LIN {X 0,Y 185.438,Z 182.881,A -85,B 0,C 180,E1 -22182.587,E2 -22182.587} C_VEL
LIN {X 0,Y 186.423,Z 185.682,A -85,B 0,C 180,E1 -22183.112,E2 -22183.112} C_VEL
LIN {X 0,Y 188.894,Z 188.498,A -85,B 0,C 180,E1 -22184.064,E2 -22184.064} C_VEL
LIN {X 0,Y 191.056,Z 191.778,A -85,B 0,C 180,E1 -22184.906,E2 -22184.906} C_VEL
LIN {X 0,Y 192.643,Z 194.162,A -85,B 0,C 180,E1 -22185.503,E2 -22185.503} C_VEL
LIN {X 0,Y 197.521,Z 201.307,A -85,B 0,C 180,E1 -22187.235,E2 -22187.235} C_VEL
LIN {X 0,Y 203.04,Z 210.464,A -85,B 0,C 180,E1 -22189.09,E2 -22189.09} C_VEL
LIN {X 0,Y 209.264,Z 223.651,A -85,B 0,C 180,E1 -22191.133,E2 -22191.133} C_VEL
LIN {X 0,Y 213.51,Z 234.001,A -85,B 0,C 180,E1 -22192.484,E2 -22192.484} C_VEL
LIN {X 0,Y 210.832,Z 286.169,A -85,B 0,C 180,E1 -22194.15,E2 -22194.15} C_VEL
LIN {X 0,Y 209.437,Z 299.447,A -85,B 0,C 180,E1 -22194.897,E2 -22194.897} C_VEL
LIN {X 0,Y 207.404,Z 312.457,A -85,B 0,C 180,E1 -22196.006,E2 -22196.006} C_VEL
LIN {X 0,Y 205.128,Z 323.758,A -85,B 0,C 180,E1 -22197.342,E2 -22197.342} C_VEL
LIN {X 0,Y 202.167,Z 335.393,A -85,B 0,C 180,E1 -22199.152,E2 -22199.152} C_VEL
LIN {X 0,Y 199.074,Z 345.843,A -85,B 0,C 180,E1 -22201.249,E2 -22201.249} C_VEL
LIN {X 0,Y 196.058,Z 355.418,A -85,B 0,C 180,E1 -22203.724,E2 -22203.724} C_VEL
LIN {X 0,Y 193.173,Z 363.626,A -85,B 0,C 180,E1 -22206.409,E2 -22206.409} C_VEL
LIN {X 0,Y 190.261,Z 371.037,A -85,B 0,C 180,E1 -22209.456,E2 -22209.456} C_VEL
LIN {X 0,Y 187.898,Z 376.982,A -85,B 0,C 180,E1 -22212.589,E2 -22212.589} C_VEL
LIN {X 0,Y 186.02,Z 381.679,A -85,B 0,C 180,E1 -22215.784,E2 -22215.784} C_VEL
LIN {X 0,Y 184.706,Z 385.27,A -85,B 0,C 180,E1 -22219.033,E2 -22219.033} C_VEL
LIN {X 0,Y 184.105,Z 387.123,A -85,B 0,C 180,E1 -22221.217,E2 -22221.217} C_VEL
LIN {X 0,Y 183.397,Z 389.328,A -85,B 0,C 180,E1 -22225.109,E2 -22225.109} C_VEL
LIN {X 0,Y 183.186,Z 390.114,A -85,B 0,C 180,E1 -22227.801,E2 -22227.801} C_VEL
LIN {X 0,Y 183.146,Z 390.342,A -85,B 0,C 180,E1 -22230,E2 -22230} C_VEL
LIN {X 0,Y 183.184,Z 390.147,A -85,B 0,C 180,E1 -22232.199,E2 -22232.199} C_VEL
LIN {X 0,Y 183.618,Z 388.592,A -85,B 0,C 180,E1 -22236.593,E2 -22236.593} C_VEL
LIN {X 0,Y 184.036,Z 387.234,A -85,B 0,C 180,E1 -22238.786,E2 -22238.786} C_VEL
LIN {X 0,Y 185.055,Z 384.362,A -85,B 0,C 180,E1 -22242.056,E2 -22242.056} C_VEL
LIN {X 0,Y 186.565,Z 380.465,A -85,B 0,C 180,E1 -22245.289,E2 -22245.289} C_VEL
LIN {X 0,Y 188.562,Z 375.438,A -85,B 0,C 180,E1 -22248.47,E2 -22248.47} C_VEL
LIN {X 0,Y 191.128,Z 369.103,A -85,B 0,C 180,E1 -22251.574,E2 -22251.574} C_VEL
LIN {X 0,Y 194.162,Z 361.178,A -85,B 0,C 180,E1 -22254.599,E2 -22254.599} C_VEL
LIN {X 0,Y 196.883,Z 353.061,A -85,B 0,C 180,E1 -22257.086,E2 -22257.086} C_VEL
LIN {X 0,Y 200.037,Z 343.242,A -85,B 0,C 180,E1 -22259.463,E2 -22259.463} C_VEL
LIN {X 0,Y 202.839,Z 333.532,A -85,B 0,C 180,E1 -22261.313,E2 -22261.313} C_VEL
LIN {X 0,Y 205.421,Z 323.01,A -85,B 0,C 180,E1 -22262.896,E2 -22262.896} C_VEL
LIN {X 0,Y 207.938,Z 310.339,A -85,B 0,C 180,E1 -22264.334,E2 -22264.334} C_VEL
LIN {X 0,Y 209.725,Z 297.869,A -85,B 0,C 180,E1 -22265.364,E2 -22265.364} C_VEL
LIN {X 0,Y 211.06,Z 284.908,A -85,B 0,C 180,E1 -22266.034,E2 -22266.034} C_VEL
LIN {X 0,Y 213.59,Z 233.928,A -85,B 0,C 180,E1 -22267.668,E2 -22267.668} C_VEL
LIN {X 0,Y 207.958,Z 220.601,A -85,B 0,C 180,E1 -22269.464,E2 -22269.464} C_VEL
LIN {X 0,Y 201.794,Z 208.024,A -85,B 0,C 180,E1 -22271.512,E2 -22271.512} C_VEL
LIN {X 0,Y 195.962,Z 198.988,A -85,B 0,C 180,E1 -22273.494,E2 -22273.494} C_VEL
LIN {X 0,Y 193.215,Z 194.973,A -85,B 0,C 180,E1 -22274.48,E2 -22274.48} C_VEL
LIN {X 0,Y 190.972,Z 191.674,A -85,B 0,C 180,E1 -22275.321,E2 -22275.321} C_VEL
LIN {X 0,Y 188.815,Z 188.335,A -85,B 0,C 180,E1 -22276.17,E2 -22276.17} C_VEL
LIN {X 0,Y 186.181,Z 185.235,A -85,B 0,C 180,E1 -22277.198,E2 -22277.198} C_VEL
LIN {X 0,Y 185.45,Z 182.877,A -85,B 0,C 180,E1 -22277.611,E2 -22277.611} C_VEL
LIN {X 0,Y 185.544,Z 182.862,A -85,B 0,C 180,E1 -22282.696,E2 -22282.696} C_VEL
LIN {X 0,Y 185.545,Z 182.864,A -85,B 0,C 180,E1 -22287.975,E2 -22287.975} C_VEL
LIN {X 0,Y 185.582,Z 182.86,A -85,B 0,C 180,E1 -22290.575,E2 -22290.575} C_VEL
LIN {X 0,Y 185.588,Z 182.867,A -85,B 0,C 180,E1 -22295.382,E2 -22295.382} C_VEL
LIN {X 0,Y 185.675,Z 182.858,A -85,B 0,C 180,E1 -22301.133,E2 -22301.133} C_VEL
LIN {X 0,Y 185.765,Z 182.842,A -85,B 0,C 180,E1 -22306.88,E2 -22306.88} C_VEL
LIN {X 0,Y 186.009,Z 182.795,A -85,B 0,C 180,E1 -22311.307,E2 -22311.307} C_VEL
LIN {X 0,Y 186.208,Z 182.773,A -85,B 0,C 180,E1 -22317.837,E2 -22317.837} C_VEL
LIN {X 0,Y 186.405,Z 182.75,A -85,B 0,C 180,E1 -22320,E2 -22320} C_VEL
LIN {X 0,Y 185.924,Z 182.815,A -85,B 0,C 180,E1 -22324.336,E2 -22324.336} C_VEL
LIN {X 0,Y 186.009,Z 182.811,A -85,B 0,C 180,E1 -22328.693,E2 -22328.693} C_VEL
LIN {X 0,Y 185.734,Z 182.829,A -85,B 0,C 180,E1 -22333.122,E2 -22333.122} C_VEL
LIN {X 0,Y 185.689,Z 182.848,A -85,B 0,C 180,E1 -22337.625,E2 -22337.625} C_VEL
LIN {X 0,Y 185.578,Z 182.868,A -85,B 0,C 180,E1 -22342.254,E2 -22342.254} C_VEL
LIN {X 0,Y 185.558,Z 182.869,A -85,B 0,C 180,E1 -22347.033,E2 -22347.033} C_VEL
LIN {X 0,Y 185.577,Z 182.86,A -85,B 0,C 180,E1 -22349.493,E2 -22349.493} C_VEL
LIN {X 0,Y 185.499,Z 182.869,A -85,B 0,C 180,E1 -22354.632,E2 -22354.632} C_VEL
LIN {X 0,Y 185.505,Z 182.874,A -85,B 0,C 180,E1 -22357.313,E2 -22357.313} C_VEL
LIN {X 0,Y 185.495,Z 183.087,A -85,B 0,C 180,E1 -22360.733,E2 -22360.733} C_VEL
LIN {X 0,Y 186.322,Z 185.835,A -85,B 0,C 180,E1 -22362.606,E2 -22362.606} C_VEL
LIN {X 0,Y 189.088,Z 190.333,A -85,B 0,C 180,E1 -22363.748,E2 -22363.748} C_VEL
LIN {X 0,Y 193.463,Z 197.495,A -85,B 0,C 180,E1 -22365.444,E2 -22365.444} C_VEL
LIN {X 0,Y 199.054,Z 207.457,A -85,B 0,C 180,E1 -22367.479,E2 -22367.479} C_VEL
LIN {X 0,Y 205.15,Z 219.677,A -85,B 0,C 180,E1 -22369.566,E2 -22369.566} C_VEL
LIN {X 0,Y 211.223,Z 234.41,A -85,B 0,C 180,E1 -22371.577,E2 -22371.577} C_VEL
LIN {X 0,Y 212.326,Z 238.091,A -85,B 0,C 180,E1 -22371.966,E2 -22371.966} C_VEL
LIN {X 0,Y 213.063,Z 245.558,A -85,B 0,C 180,E1 -22372.431,E2 -22372.431} C_VEL
LIN {X 0,Y 212.354,Z 259.49,A -85,B 0,C 180,E1 -22372.865,E2 -22372.865} C_VEL
LIN {X 0,Y 211.584,Z 265.346,A -85,B 0,C 180,E1 -22372.946,E2 -22372.946} C_VEL
LIN {X 0,Y 205.962,Z 284.372,A -85,B 0,C 180,E1 -22372.571,E2 -22372.571} C_VEL
LIN {X 0,Y 205.095,Z 290.216,A -85,B 0,C 180,E1 -22372.672,E2 -22372.672} C_VEL
LIN {X 0,Y 203.834,Z 303.973,A -85,B 0,C 180,E1 -22373.356,E2 -22373.356} C_VEL
LIN {X 0,Y 201.749,Z 316.536,A -85,B 0,C 180,E1 -22374.304,E2 -22374.304} C_VEL
LIN {X 0,Y 199.213,Z 328.676,A -85,B 0,C 180,E1 -22375.635,E2 -22375.635} C_VEL
LIN {X 0,Y 196.423,Z 339.649,A -85,B 0,C 180,E1 -22377.237,E2 -22377.237} C_VEL
LIN {X 0,Y 192.952,Z 350.849,A -85,B 0,C 180,E1 -22379.341,E2 -22379.341} C_VEL
LIN {X 0,Y 189.536,Z 360.785,A -85,B 0,C 180,E1 -22381.786,E2 -22381.786} C_VEL
LIN {X 0,Y 186.521,Z 368.936,A -85,B 0,C 180,E1 -22384.322,E2 -22384.322} C_VEL
LIN {X 0,Y 183.553,Z 376.941,A -85,B 0,C 180,E1 -22387.488,E2 -22387.488} C_VEL
LIN {X 0,Y 180.921,Z 383.353,A -85,B 0,C 180,E1 -22390.72,E2 -22390.72} C_VEL
LIN {X 0,Y 178.761,Z 388.446,A -85,B 0,C 180,E1 -22394.026,E2 -22394.026} C_VEL
LIN {X 0,Y 177.39,Z 392.408,A -85,B 0,C 180,E1 -22397.414,E2 -22397.414} C_VEL
LIN {X 0,Y 176.468,Z 395.337,A -85,B 0,C 180,E1 -22400.834,E2 -22400.834} C_VEL
LIN {X 0,Y 175.946,Z 397.726,A -85,B 0,C 180,E1 -22405.418,E2 -22405.418} C_VEL
LIN {X 0,Y 175.949,Z 398.335,A -85,B 0,C 180,E1 -22407.711,E2 -22407.711} C_VEL
LIN {X 0,Y 176.022,Z 398.547,A -85,B 0,C 180,E1 -22410,E2 -22410} C_VEL
LIN {X 0,Y 175.947,Z 398.162,A -85,B 0,C 180,E1 -22413.037,E2 -22413.037} C_VEL
LIN {X 0,Y 176.137,Z 396.699,A -85,B 0,C 180,E1 -22416.875,E2 -22416.875} C_VEL
LIN {X 0,Y 176.468,Z 395.291,A -85,B 0,C 180,E1 -22419.167,E2 -22419.167} C_VEL
LIN {X 0,Y 177.39,Z 392.343,A -85,B 0,C 180,E1 -22422.586,E2 -22422.586} C_VEL
LIN {X 0,Y 178.76,Z 388.356,A -85,B 0,C 180,E1 -22425.974,E2 -22425.974} C_VEL
LIN {X 0,Y 181.33,Z 382.235,A -85,B 0,C 180,E1 -22429.824,E2 -22429.824} C_VEL
LIN {X 0,Y 184.328,Z 374.773,A -85,B 0,C 180,E1 -22433.379,E2 -22433.379} C_VEL
LIN {X 0,Y 187.075,Z 367.259,A -85,B 0,C 180,E1 -22436.195,E2 -22436.195} C_VEL
LIN {X 0,Y 190.171,Z 358.756,A -85,B 0,C 180,E1 -22438.713,E2 -22438.713} C_VEL
LIN {X 0,Y 193.689,Z 348.253,A -85,B 0,C 180,E1 -22441.135,E2 -22441.135} C_VEL
LIN {X 0,Y 197.144,Z 336.428,A -85,B 0,C 180,E1 -22443.237,E2 -22443.237} C_VEL
LIN {X 0,Y 200.028,Z 324.506,A -85,B 0,C 180,E1 -22444.816,E2 -22444.816} C_VEL
LIN {X 0,Y 202.45,Z 312.094,A -85,B 0,C 180,E1 -22446.014,E2 -22446.014} C_VEL
LIN {X 0,Y 204.293,Z 299.341,A -85,B 0,C 180,E1 -22446.856,E2 -22446.856} C_VEL
LIN {X 0,Y 205.334,Z 285.462,A -85,B 0,C 180,E1 -22447.419,E2 -22447.419} C_VEL
LIN {X 0,Y 207.266,Z 245.004,A -85,B 0,C 180,E1 -22448.75,E2 -22448.75} C_VEL
LIN {X 0,Y 206.492,Z 239.162,A -85,B 0,C 180,E1 -22449.177,E2 -22449.177} C_VEL
LIN {X 0,Y 201.216,Z 225.726,A -85,B 0,C 180,E1 -22451.022,E2 -22451.022} C_VEL
LIN {X 0,Y 195.205,Z 212.97,A -85,B 0,C 180,E1 -22453.19,E2 -22453.19} C_VEL
LIN {X 0,Y 188.351,Z 200.534,A -85,B 0,C 180,E1 -22455.828,E2 -22455.828} C_VEL
LIN {X 0,Y 183.78,Z 193.268,A -85,B 0,C 180,E1 -22457.716,E2 -22457.716} C_VEL
LIN {X 0,Y 181.859,Z 190.145,A -85,B 0,C 180,E1 -22458.563,E2 -22458.563} C_VEL
LIN {X 0,Y 178.959,Z 185.72,A -85,B 0,C 180,E1 -22459.887,E2 -22459.887} C_VEL
LIN {X 0,Y 178.665,Z 184.95,A -85,B 0,C 180,E1 -22460.267,E2 -22460.267} C_VEL
LIN {X 0,Y 178.412,Z 183.762,A -85,B 0,C 180,E1 -22461.242,E2 -22461.242} C_VEL
LIN {X 0,Y 178.484,Z 183.753,A -85,B 0,C 180,E1 -22466.546,E2 -22466.546} C_VEL
LIN {X 0,Y 178.444,Z 183.752,A -85,B 0,C 180,E1 -22471.796,E2 -22471.796} C_VEL
LIN {X 0,Y 178.516,Z 183.749,A -85,B 0,C 180,E1 -22474.889,E2 -22474.889} C_VEL
LIN {X 0,Y 178.623,Z 183.731,A -85,B 0,C 180,E1 -22480.785,E2 -22480.785} C_VEL
LIN {X 0,Y 178.658,Z 183.724,A -85,B 0,C 180,E1 -22486.348,E2 -22486.348} C_VEL
LIN {X 0,Y 178.912,Z 183.7,A -85,B 0,C 180,E1 -22490.96,E2 -22490.96} C_VEL
LIN {X 0,Y 179.153,Z 183.664,A -85,B 0,C 180,E1 -22497.752,E2 -22497.752} C_VEL
LIN {X 0,Y 179.369,Z 183.629,A -85,B 0,C 180,E1 -22500,E2 -22500} C_VEL
LIN {X 0,Y 178.867,Z 183.694,A -85,B 0,C 180,E1 -22504.507,E2 -22504.507} C_VEL
LIN {X 0,Y 178.912,Z 183.699,A -85,B 0,C 180,E1 -22509.04,E2 -22509.04} C_VEL
LIN {X 0,Y 178.659,Z 183.729,A -85,B 0,C 180,E1 -22513.652,E2 -22513.652} C_VEL
LIN {X 0,Y 178.639,Z 183.731,A -85,B 0,C 180,E1 -22519.23,E2 -22519.23} C_VEL
LIN {X 0,Y 178.535,Z 183.746,A -85,B 0,C 180,E1 -22525.125,E2 -22525.125} C_VEL
LIN {X 0,Y 178.48,Z 183.749,A -85,B 0,C 180,E1 -22530.791,E2 -22530.791} C_VEL
LIN {X 0,Y 178.493,Z 183.752,A -85,B 0,C 180,E1 -22534.223,E2 -22534.223} C_VEL
LIN {X 0,Y 178.43,Z 183.754,A -85,B 0,C 180,E1 -22539.796,E2 -22539.796} C_VEL
LIN {X 0,Y 178.447,Z 183.753,A -85,B 0,C 180,E1 -22540.16,E2 -22540.16} C_VEL
LIN {X 0,Y 179.378,Z 186.499,A -85,B 0,C 180,E1 -22540.684,E2 -22540.684} C_VEL
LIN {X 0,Y 181.415,Z 188.713,A -85,B 0,C 180,E1 -22541.562,E2 -22541.562} C_VEL
LIN {X 0,Y 184.268,Z 192.886,A -85,B 0,C 180,E1 -22542.795,E2 -22542.795} C_VEL
LIN {X 0,Y 185.614,Z 194.718,A -85,B 0,C 180,E1 -22543.346,E2 -22543.346} C_VEL
LIN {X 0,Y 188.82,Z 199.398,A -85,B 0,C 180,E1 -22544.623,E2 -22544.623} C_VEL
LIN {X 0,Y 195.085,Z 208.87,A -85,B 0,C 180,E1 -22546.94,E2 -22546.94} C_VEL
LIN {X 0,Y 199.32,Z 216.409,A -85,B 0,C 180,E1 -22548.433,E2 -22548.433} C_VEL
LIN {X 0,Y 206.254,Z 231.957,A -85,B 0,C 180,E1 -22550.819,E2 -22550.819} C_VEL
LIN {X 0,Y 207.807,Z 235.855,A -85,B 0,C 180,E1 -22551.339,E2 -22551.339} C_VEL
LIN {X 0,Y 205.268,Z 284.588,A -85,B 0,C 180,E1 -22552.926,E2 -22552.926} C_VEL
LIN {X 0,Y 203.962,Z 297.662,A -85,B 0,C 180,E1 -22553.612,E2 -22553.612} C_VEL
LIN {X 0,Y 202.37,Z 308.094,A -85,B 0,C 180,E1 -22554.43,E2 -22554.43} C_VEL
LIN {X 0,Y 199.971,Z 320.431,A -85,B 0,C 180,E1 -22555.784,E2 -22555.784} C_VEL
LIN {X 0,Y 197.266,Z 331.509,A -85,B 0,C 180,E1 -22557.394,E2 -22557.394} C_VEL
LIN {X 0,Y 193.921,Z 342.804,A -85,B 0,C 180,E1 -22559.51,E2 -22559.51} C_VEL
LIN {X 0,Y 190.885,Z 352.098,A -85,B 0,C 180,E1 -22561.777,E2 -22561.777} C_VEL
LIN {X 0,Y 187.801,Z 360.925,A -85,B 0,C 180,E1 -22564.51,E2 -22564.51} C_VEL
LIN {X 0,Y 184.585,Z 368.922,A -85,B 0,C 180,E1 -22567.62,E2 -22567.62} C_VEL
LIN {X 0,Y 181.882,Z 375.338,A -85,B 0,C 180,E1 -22570.826,E2 -22570.826} C_VEL
LIN {X 0,Y 179.745,Z 380.425,A -85,B 0,C 180,E1 -22574.115,E2 -22574.115} C_VEL
LIN {X 0,Y 178.15,Z 384.373,A -85,B 0,C 180,E1 -22577.469,E2 -22577.469} C_VEL
LIN {X 0,Y 177.084,Z 387.286,A -85,B 0,C 180,E1 -22580.866,E2 -22580.866} C_VEL
LIN {X 0,Y 176.568,Z 388.678,A -85,B 0,C 180,E1 -22583.142,E2 -22583.142} C_VEL
LIN {X 0,Y 176.262,Z 389.668,A -85,B 0,C 180,E1 -22585.426,E2 -22585.426} C_VEL
LIN {X 0,Y 176.102,Z 390.276,A -85,B 0,C 180,E1 -22587.713,E2 -22587.713} C_VEL
LIN {X 0,Y 176.058,Z 390.504,A -85,B 0,C 180,E1 -22590,E2 -22590} C_VEL
LIN {X 0,Y 176.1,Z 390.309,A -85,B 0,C 180,E1 -22592.287,E2 -22592.287} C_VEL
LIN {X 0,Y 176.562,Z 388.754,A -85,B 0,C 180,E1 -22596.858,E2 -22596.858} C_VEL
LIN {X 0,Y 177.033,Z 387.395,A -85,B 0,C 180,E1 -22599.137,E2 -22599.137} C_VEL
LIN {X 0,Y 178.12,Z 384.523,A -85,B 0,C 180,E1 -22602.533,E2 -22602.533} C_VEL
LIN {X 0,Y 179.718,Z 380.626,A -85,B 0,C 180,E1 -22605.887,E2 -22605.887} C_VEL
LIN {X 0,Y 181.834,Z 375.599,A -85,B 0,C 180,E1 -22609.179,E2 -22609.179} C_VEL
LIN {X 0,Y 184.544,Z 369.263,A -85,B 0,C 180,E1 -22612.385,E2 -22612.385} C_VEL
LIN {X 0,Y 187.71,Z 361.338,A -85,B 0,C 180,E1 -22615.503,E2 -22615.503} C_VEL
LIN {X 0,Y 190.575,Z 353.263,A -85,B 0,C 180,E1 -22618.046,E2 -22618.046} C_VEL
LIN {X 0,Y 193.884,Z 343.4,A -85,B 0,C 180,E1 -22620.496,E2 -22620.496} C_VEL
LIN {X 0,Y 196.825,Z 333.689,A -85,B 0,C 180,E1 -22622.385,E2 -22622.385} C_VEL
LIN {X 0,Y 199.494,Z 323.167,A -85,B 0,C 180,E1 -22624.004,E2 -22624.004} C_VEL
LIN {X 0,Y 202.127,Z 310.494,A -85,B 0,C 180,E1 -22625.466,E2 -22625.466} C_VEL
LIN {X 0,Y 204.024,Z 297.735,A -85,B 0,C 180,E1 -22626.538,E2 -22626.538} C_VEL
LIN {X 0,Y 205.354,Z 285.32,A -85,B 0,C 180,E1 -22627.187,E2 -22627.187} C_VEL
LIN {X 0,Y 207.85,Z 235.79,A -85,B 0,C 180,E1 -22628.824,E2 -22628.824} C_VEL
LIN {X 0,Y 201.999,Z 221.957,A -85,B 0,C 180,E1 -22630.814,E2 -22630.814} C_VEL
LIN {X 0,Y 196.888,Z 211.745,A -85,B 0,C 180,E1 -22632.613,E2 -22632.613} C_VEL
LIN {X 0,Y 190.234,Z 201.344,A -85,B 0,C 180,E1 -22635.038,E2 -22635.038} C_VEL
LIN {X 0,Y 184.437,Z 193.04,A -85,B 0,C 180,E1 -22637.346,E2 -22637.346} C_VEL
LIN {X 0,Y 182.218,Z 189.939,A -85,B 0,C 180,E1 -22638.293,E2 -22638.293} C_VEL
LIN {X 0,Y 181.458,Z 188.733,A -85,B 0,C 180,E1 -22638.635,E2 -22638.635} C_VEL
LIN {X 0,Y 179.398,Z 186.531,A -85,B 0,C 180,E1 -22639.525,E2 -22639.525} C_VEL
LIN {X 0,Y 178.453,Z 183.756,A -85,B 0,C 180,E1 -22640.118,E2 -22640.118} C_VEL
LIN {X 0,Y 178.496,Z 183.738,A -85,B 0,C 180,E1 -22645.775,E2 -22645.775} C_VEL
LIN {X 0,Y 178.523,Z 183.744,A -85,B 0,C 180,E1 -22650.006,E2 -22650.006} C_VEL
LIN {X 0,Y 178.535,Z 183.746,A -85,B 0,C 180,E1 -22654.875,E2 -22654.875} C_VEL
LIN {X 0,Y 178.624,Z 183.735,A -85,B 0,C 180,E1 -22660.784,E2 -22660.784} C_VEL
LIN {X 0,Y 178.682,Z 183.72,A -85,B 0,C 180,E1 -22666.35,E2 -22666.35} C_VEL
LIN {X 0,Y 178.938,Z 183.675,A -85,B 0,C 180,E1 -22670.961,E2 -22670.961} C_VEL
LIN {X 0,Y 179.154,Z 183.651,A -85,B 0,C 180,E1 -22677.752,E2 -22677.752} C_VEL
LIN {X 0,Y 179.368,Z 183.626,A -85,B 0,C 180,E1 -22680,E2 -22680} C_VEL
LIN {X 0,Y 178.872,Z 183.691,A -85,B 0,C 180,E1 -22684.507,E2 -22684.507} C_VEL
LIN {X 0,Y 178.959,Z 183.692,A -85,B 0,C 180,E1 -22689.038,E2 -22689.038} C_VEL
LIN {X 0,Y 178.666,Z 183.709,A -85,B 0,C 180,E1 -22693.651,E2 -22693.651} C_VEL
LIN {X 0,Y 178.649,Z 183.718,A -85,B 0,C 180,E1 -22698.344,E2 -22698.344} C_VEL
LIN {X 0,Y 178.497,Z 183.749,A -85,B 0,C 180,E1 -22703.187,E2 -22703.187} C_VEL
LIN {X 0,Y 178.485,Z 183.752,A -85,B 0,C 180,E1 -22708.197,E2 -22708.197} C_VEL
LIN {X 0,Y 178.477,Z 183.743,A -85,B 0,C 180,E1 -22710.791,E2 -22710.791} C_VEL
LIN {X 0,Y 178.484,Z 183.743,A -85,B 0,C 180,E1 -22714.219,E2 -22714.219} C_VEL
LIN {X 0,Y 178.417,Z 183.872,A -85,B 0,C 180,E1 -22718.757,E2 -22718.757} C_VEL
LIN {X 0,Y 178.895,Z 185.52,A -85,B 0,C 180,E1 -22719.947,E2 -22719.947} C_VEL
LIN {X 0,Y 181.77,Z 190.049,A -85,B 0,C 180,E1 -22721.278,E2 -22721.278} C_VEL
LIN {X 0,Y 183.051,Z 192.016,A -85,B 0,C 180,E1 -22721.843,E2 -22721.843} C_VEL
LIN {X 0,Y 187.094,Z 198.569,A -85,B 0,C 180,E1 -22723.559,E2 -22723.559} C_VEL
LIN {X 0,Y 191.402,Z 205.843,A -85,B 0,C 180,E1 -22725.269,E2 -22725.269} C_VEL
LIN {X 0,Y 197.565,Z 217.59,A -85,B 0,C 180,E1 -22727.574,E2 -22727.574} C_VEL
LIN {X 0,Y 203.143,Z 230.178,A -85,B 0,C 180,E1 -22729.563,E2 -22729.563} C_VEL
LIN {X 0,Y 206.773,Z 239.68,A -85,B 0,C 180,E1 -22730.828,E2 -22730.828} C_VEL
LIN {X 0,Y 207.444,Z 245.987,A -85,B 0,C 180,E1 -22731.252,E2 -22731.252} C_VEL
LIN {X 0,Y 205.095,Z 290.216,A -85,B 0,C 180,E1 -22732.672,E2 -22732.672} C_VEL
LIN {X 0,Y 204.558,Z 294.107,A -85,B 0,C 180,E1 -22732.764,E2 -22732.764} C_VEL
LIN {X 0,Y 202.211,Z 301.678,A -85,B 0,C 180,E1 -22732.816,E2 -22732.816} C_VEL
LIN {X 0,Y 196.875,Z 314.527,A -85,B 0,C 180,E1 -22733.032,E2 -22733.032} C_VEL
LIN {X 0,Y 195.298,Z 320.024,A -85,B 0,C 180,E1 -22733.452,E2 -22733.452} C_VEL
LIN {X 0,Y 192.536,Z 331.95,A -85,B 0,C 180,E1 -22734.907,E2 -22734.907} C_VEL
LIN {X 0,Y 189.274,Z 343.502,A -85,B 0,C 180,E1 -22736.792,E2 -22736.792} C_VEL
LIN {X 0,Y 185.763,Z 353.904,A -85,B 0,C 180,E1 -22738.971,E2 -22738.971} C_VEL
LIN {X 0,Y 182.615,Z 362.41,A -85,B 0,C 180,E1 -22741.245,E2 -22741.245} C_VEL
LIN {X 0,Y 179.56,Z 370.262,A -85,B 0,C 180,E1 -22743.875,E2 -22743.875} C_VEL
LIN {X 0,Y 176.475,Z 377.933,A -85,B 0,C 180,E1 -22747.152,E2 -22747.152} C_VEL
LIN {X 0,Y 173.385,Z 385.01,A -85,B 0,C 180,E1 -22751.079,E2 -22751.079} C_VEL
LIN {X 0,Y 171.351,Z 389.717,A -85,B 0,C 180,E1 -22754.538,E2 -22754.538} C_VEL
LIN {X 0,Y 170.053,Z 393.318,A -85,B 0,C 180,E1 -22758.075,E2 -22758.075} C_VEL
LIN {X 0,Y 169.427,Z 395.174,A -85,B 0,C 180,E1 -22760.449,E2 -22760.449} C_VEL
LIN {X 0,Y 168.86,Z 397.564,A -85,B 0,C 180,E1 -22765.225,E2 -22765.225} C_VEL
LIN {X 0,Y 168.858,Z 398.173,A -85,B 0,C 180,E1 -22767.615,E2 -22767.615} C_VEL
LIN {X 0,Y 168.934,Z 398.385,A -85,B 0,C 180,E1 -22770,E2 -22770} C_VEL
LIN {X 0,Y 168.85,Z 398.109,A -85,B 0,C 180,E1 -22772.627,E2 -22772.627} C_VEL
LIN {X 0,Y 169.072,Z 396.536,A -85,B 0,C 180,E1 -22777.164,E2 -22777.164} C_VEL
LIN {X 0,Y 169.427,Z 395.128,A -85,B 0,C 180,E1 -22779.551,E2 -22779.551} C_VEL
LIN {X 0,Y 170.436,Z 392.179,A -85,B 0,C 180,E1 -22783.109,E2 -22783.109} C_VEL
LIN {X 0,Y 171.92,Z 388.192,A -85,B 0,C 180,E1 -22786.628,E2 -22786.628} C_VEL
LIN {X 0,Y 174.637,Z 382.071,A -85,B 0,C 180,E1 -22790.618,E2 -22790.618} C_VEL
LIN {X 0,Y 177.485,Z 375.379,A -85,B 0,C 180,E1 -22793.95,E2 -22793.95} C_VEL
LIN {X 0,Y 180.691,Z 367.093,A -85,B 0,C 180,E1 -22797.195,E2 -22797.195} C_VEL
LIN {X 0,Y 183.952,Z 358.59,A -85,B 0,C 180,E1 -22799.78,E2 -22799.78} C_VEL
LIN {X 0,Y 187.638,Z 348.087,A -85,B 0,C 180,E1 -22802.258,E2 -22802.258} C_VEL
LIN {X 0,Y 191.245,Z 336.262,A -85,B 0,C 180,E1 -22804.403,E2 -22804.403} C_VEL
LIN {X 0,Y 194.236,Z 324.338,A -85,B 0,C 180,E1 -22806.013,E2 -22806.013} C_VEL
LIN {X 0,Y 196.743,Z 311.924,A -85,B 0,C 180,E1 -22807.231,E2 -22807.231} C_VEL
LIN {X 0,Y 198.665,Z 299.183,A -85,B 0,C 180,E1 -22808.081,E2 -22808.081} C_VEL
LIN {X 0,Y 199.793,Z 284.339,A -85,B 0,C 180,E1 -22808.687,E2 -22808.687} C_VEL
LIN {X 0,Y 201.734,Z 246.08,A -85,B 0,C 180,E1 -22809.965,E2 -22809.965} C_VEL
LIN {X 0,Y 201.101,Z 241.562,A -85,B 0,C 180,E1 -22810.321,E2 -22810.321} C_VEL
LIN {X 0,Y 195.466,Z 227.242,A -85,B 0,C 180,E1 -22812.421,E2 -22812.421} C_VEL
LIN {X 0,Y 189.097,Z 214.028,A -85,B 0,C 180,E1 -22814.887,E2 -22814.887} C_VEL
LIN {X 0,Y 183.283,Z 203.692,A -85,B 0,C 180,E1 -22817.294,E2 -22817.294} C_VEL
LIN {X 0,Y 178.309,Z 195.507,A -85,B 0,C 180,E1 -22819.537,E2 -22819.537} C_VEL
LIN {X 0,Y 174.548,Z 189.931,A -85,B 0,C 180,E1 -22821.354,E2 -22821.354} C_VEL
LIN {X 0,Y 172.188,Z 187.163,A -85,B 0,C 180,E1 -22822.525,E2 -22822.525} C_VEL
LIN {X 0,Y 171.415,Z 184.96,A -85,B 0,C 180,E1 -22823.065,E2 -22823.065} C_VEL
LIN {X 0,Y 171.381,Z 184.637,A -85,B 0,C 180,E1 -22823.515,E2 -22823.515} C_VEL
LIN {X 0,Y 171.418,Z 184.632,A -85,B 0,C 180,E1 -22829.427,E2 -22829.427} C_VEL
LIN {X 0,Y 171.444,Z 184.628,A -85,B 0,C 180,E1 -22834.402,E2 -22834.402} C_VEL
LIN {X 0,Y 171.579,Z 184.606,A -85,B 0,C 180,E1 -22840.872,E2 -22840.872} C_VEL
LIN {X 0,Y 171.577,Z 184.61,A -85,B 0,C 180,E1 -22845.773,E2 -22845.773} C_VEL
LIN {X 0,Y 171.849,Z 184.579,A -85,B 0,C 180,E1 -22850.585,E2 -22850.585} C_VEL
LIN {X 0,Y 171.817,Z 184.578,A -85,B 0,C 180,E1 -22855.308,E2 -22855.308} C_VEL
LIN {X 0,Y 172.332,Z 184.505,A -85,B 0,C 180,E1 -22860,E2 -22860} C_VEL
LIN {X 0,Y 171.815,Z 184.57,A -85,B 0,C 180,E1 -22864.693,E2 -22864.693} C_VEL
LIN {X 0,Y 171.849,Z 184.577,A -85,B 0,C 180,E1 -22869.415,E2 -22869.415} C_VEL
LIN {X 0,Y 171.58,Z 184.612,A -85,B 0,C 180,E1 -22874.227,E2 -22874.227} C_VEL
LIN {X 0,Y 171.559,Z 184.615,A -85,B 0,C 180,E1 -22879.575,E2 -22879.575} C_VEL
LIN {X 0,Y 171.47,Z 184.626,A -85,B 0,C 180,E1 -22885.617,E2 -22885.617} C_VEL
LIN {X 0,Y 171.443,Z 184.626,A -85,B 0,C 180,E1 -22890.587,E2 -22890.587} C_VEL
LIN {X 0,Y 171.403,Z 184.628,A -85,B 0,C 180,E1 -22896.48,E2 -22896.48} C_VEL
LIN {X 0,Y 171.396,Z 184.634,A -85,B 0,C 180,E1 -22897.308,E2 -22897.308} C_VEL
LIN {X 0,Y 172.287,Z 187.267,A -85,B 0,C 180,E1 -22897.891,E2 -22897.891} C_VEL
LIN {X 0,Y 174.275,Z 189.515,A -85,B 0,C 180,E1 -22898.873,E2 -22898.873} C_VEL
LIN {X 0,Y 175.154,Z 190.413,A -85,B 0,C 180,E1 -22899.288,E2 -22899.288} C_VEL
LIN {X 0,Y 177.244,Z 193.633,A -85,B 0,C 180,E1 -22900.311,E2 -22900.311} C_VEL
LIN {X 0,Y 178.639,Z 195.287,A -85,B 0,C 180,E1 -22900.939,E2 -22900.939} C_VEL
LIN {X 0,Y 181.349,Z 199.009,A -85,B 0,C 180,E1 -22902.139,E2 -22902.139} C_VEL
LIN {X 0,Y 189.231,Z 210.901,A -85,B 0,C 180,E1 -22905.356,E2 -22905.356} C_VEL
LIN {X 0,Y 194.301,Z 219.723,A -85,B 0,C 180,E1 -22907.262,E2 -22907.262} C_VEL
LIN {X 0,Y 200.847,Z 234.43,A -85,B 0,C 180,E1 -22909.656,E2 -22909.656} C_VEL
LIN {X 0,Y 202.22,Z 237.907,A -85,B 0,C 180,E1 -22910.146,E2 -22910.146} C_VEL
LIN {X 0,Y 199.625,Z 285.168,A -85,B 0,C 180,E1 -22911.714,E2 -22911.714} C_VEL
LIN {X 0,Y 198.269,Z 298.107,A -85,B 0,C 180,E1 -22912.419,E2 -22912.419} C_VEL
LIN {X 0,Y 196.643,Z 308.264,A -85,B 0,C 180,E1 -22913.227,E2 -22913.227} C_VEL
LIN {X 0,Y 194.154,Z 320.598,A -85,B 0,C 180,E1 -22914.608,E2 -22914.608} C_VEL
LIN {X 0,Y 191.325,Z 331.675,A -85,B 0,C 180,E1 -22916.249,E2 -22916.249} C_VEL
LIN {X 0,Y 187.833,Z 342.97,A -85,B 0,C 180,E1 -22918.411,E2 -22918.411} C_VEL
LIN {X 0,Y 184.405,Z 352.935,A -85,B 0,C 180,E1 -22920.928,E2 -22920.928} C_VEL
LIN {X 0,Y 180.88,Z 362.568,A -85,B 0,C 180,E1 -22924.08,E2 -22924.08} C_VEL
LIN {X 0,Y 177.552,Z 370.253,A -85,B 0,C 180,E1 -22927.298,E2 -22927.298} C_VEL
LIN {X 0,Y 174.356,Z 377.31,A -85,B 0,C 180,E1 -22931.188,E2 -22931.188} C_VEL
LIN {X 0,Y 172.277,Z 382.006,A -85,B 0,C 180,E1 -22934.623,E2 -22934.623} C_VEL
LIN {X 0,Y 170.764,Z 385.596,A -85,B 0,C 180,E1 -22938.125,E2 -22938.125} C_VEL
LIN {X 0,Y 170.069,Z 387.449,A -85,B 0,C 180,E1 -22940.485,E2 -22940.485} C_VEL
LIN {X 0,Y 169.526,Z 388.841,A -85,B 0,C 180,E1 -22942.856,E2 -22942.856} C_VEL
LIN {X 0,Y 169.007,Z 390.439,A -85,B 0,C 180,E1 -22947.617,E2 -22947.617} C_VEL
LIN {X 0,Y 168.972,Z 390.666,A -85,B 0,C 180,E1 -22950,E2 -22950} C_VEL
LIN {X 0,Y 169.134,Z 390.063,A -85,B 0,C 180,E1 -22954.229,E2 -22954.229} C_VEL
LIN {X 0,Y 169.52,Z 388.915,A -85,B 0,C 180,E1 -22957.145,E2 -22957.145} C_VEL
LIN {X 0,Y 170.01,Z 387.557,A -85,B 0,C 180,E1 -22959.518,E2 -22959.518} C_VEL
LIN {X 0,Y 171.178,Z 384.685,A -85,B 0,C 180,E1 -22963.05,E2 -22963.05} C_VEL
LIN {X 0,Y 172.899,Z 380.787,A -85,B 0,C 180,E1 -22966.531,E2 -22966.531} C_VEL
LIN {X 0,Y 175.141,Z 375.759,A -85,B 0,C 180,E1 -22969.943,E2 -22969.943} C_VEL
LIN {X 0,Y 178.005,Z 369.423,A -85,B 0,C 180,E1 -22973.255,E2 -22973.255} C_VEL
LIN {X 0,Y 181.24,Z 361.694,A -85,B 0,C 180,E1 -22976.401,E2 -22976.401} C_VEL
LIN {X 0,Y 184.334,Z 353.422,A -85,B 0,C 180,E1 -22979.085,E2 -22979.085} C_VEL
LIN {X 0,Y 187.813,Z 343.559,A -85,B 0,C 180,E1 -22981.593,E2 -22981.593} C_VEL
LIN {X 0,Y 190.873,Z 333.847,A -85,B 0,C 180,E1 -22983.525,E2 -22983.525} C_VEL
LIN {X 0,Y 193.655,Z 323.323,A -85,B 0,C 180,E1 -22985.178,E2 -22985.178} C_VEL
LIN {X 0,Y 196.397,Z 310.648,A -85,B 0,C 180,E1 -22986.666,E2 -22986.666} C_VEL
LIN {X 0,Y 198.332,Z 298.219,A -85,B 0,C 180,E1 -22987.731,E2 -22987.731} C_VEL
LIN {X 0,Y 199.731,Z 285.725,A -85,B 0,C 180,E1 -22988.407,E2 -22988.407} C_VEL
LIN {X 0,Y 202.265,Z 237.923,A -85,B 0,C 180,E1 -22990.019,E2 -22990.019} C_VEL
LIN {X 0,Y 197.086,Z 225.556,A -85,B 0,C 180,E1 -22991.893,E2 -22991.893} C_VEL
LIN {X 0,Y 192.557,Z 216.344,A -85,B 0,C 180,E1 -22993.583,E2 -22993.583} C_VEL
LIN {X 0,Y 186.433,Z 206.562,A -85,B 0,C 180,E1 -22995.941,E2 -22995.941} C_VEL
LIN {X 0,Y 180.722,Z 198.314,A -85,B 0,C 180,E1 -22998.337,E2 -22998.337} C_VEL
LIN {X 0,Y 177.858,Z 194.233,A -85,B 0,C 180,E1 -22999.639,E2 -22999.639} C_VEL
LIN {X 0,Y 175.626,Z 191.295,A -85,B 0,C 180,E1 -23000.694,E2 -23000.694} C_VEL
LIN {X 0,Y 174.797,Z 189.854,A -85,B 0,C 180,E1 -23001.121,E2 -23001.121} C_VEL
LIN {X 0,Y 172.586,Z 187.733,A -85,B 0,C 180,E1 -23002.186,E2 -23002.186} C_VEL
LIN {X 0,Y 171.519,Z 185.307,A -85,B 0,C 180,E1 -23002.815,E2 -23002.815} C_VEL
LIN {X 0,Y 171.405,Z 184.623,A -85,B 0,C 180,E1 -23002.971,E2 -23002.971} C_VEL
LIN {X 0,Y 171.428,Z 184.619,A -85,B 0,C 180,E1 -23007.794,E2 -23007.794} C_VEL
LIN {X 0,Y 171.449,Z 184.619,A -85,B 0,C 180,E1 -23010.534,E2 -23010.534} C_VEL
LIN {X 0,Y 171.458,Z 184.624,A -85,B 0,C 180,E1 -23015.801,E2 -23015.801} C_VEL
LIN {X 0,Y 171.58,Z 184.612,A -85,B 0,C 180,E1 -23020.872,E2 -23020.872} C_VEL
LIN {X 0,Y 171.594,Z 184.595,A -85,B 0,C 180,E1 -23025.774,E2 -23025.774} C_VEL
LIN {X 0,Y 171.873,Z 184.556,A -85,B 0,C 180,E1 -23030.586,E2 -23030.586} C_VEL
LIN {X 0,Y 171.823,Z 184.582,A -85,B 0,C 180,E1 -23035.308,E2 -23035.308} C_VEL
LIN {X 0,Y 172.331,Z 184.501,A -85,B 0,C 180,E1 -23040,E2 -23040} C_VEL
LIN {X 0,Y 171.821,Z 184.567,A -85,B 0,C 180,E1 -23044.692,E2 -23044.692} C_VEL
LIN {X 0,Y 171.888,Z 184.573,A -85,B 0,C 180,E1 -23049.413,E2 -23049.413} C_VEL
LIN {X 0,Y 171.593,Z 184.593,A -85,B 0,C 180,E1 -23054.226,E2 -23054.226} C_VEL
LIN {X 0,Y 171.54,Z 184.598,A -85,B 0,C 180,E1 -23059.558,E2 -23059.558} C_VEL
LIN {X 0,Y 171.458,Z 184.613,A -85,B 0,C 180,E1 -23065.609,E2 -23065.609} C_VEL
LIN {X 0,Y 171.44,Z 184.619,A -85,B 0,C 180,E1 -23070.586,E2 -23070.586} C_VEL
LIN {X 0,Y 171.378,Z 184.646,A -85,B 0,C 180,E1 -23076.532,E2 -23076.532} C_VEL
LIN {X 0,Y 171.428,Z 185.016,A -85,B 0,C 180,E1 -23076.84,E2 -23076.84} C_VEL
LIN {X 0,Y 172.371,Z 187.483,A -85,B 0,C 180,E1 -23077.428,E2 -23077.428} C_VEL
LIN {X 0,Y 175.783,Z 191.623,A -85,B 0,C 180,E1 -23079.114,E2 -23079.114} C_VEL
LIN {X 0,Y 179.96,Z 198.211,A -85,B 0,C 180,E1 -23081.106,E2 -23081.106} C_VEL
LIN {X 0,Y 182.934,Z 203.033,A -85,B 0,C 180,E1 -23082.432,E2 -23082.432} C_VEL
LIN {X 0,Y 187.872,Z 211.743,A -85,B 0,C 180,E1 -23084.513,E2 -23084.513} C_VEL
LIN {X 0,Y 193.556,Z 222.981,A -85,B 0,C 180,E1 -23086.754,E2 -23086.754} C_VEL
LIN {X 0,Y 198.813,Z 235.205,A -85,B 0,C 180,E1 -23088.733,E2 -23088.733} C_VEL
LIN {X 0,Y 201.49,Z 242.558,A -85,B 0,C 180,E1 -23089.731,E2 -23089.731} C_VEL
LIN {X 0,Y 201.867,Z 247.666,A -85,B 0,C 180,E1 -23090.053,E2 -23090.053} C_VEL
LIN {X 0,Y 199.159,Z 294.791,A -85,B 0,C 180,E1 -23091.633,E2 -23091.633} C_VEL
LIN {X 0,Y 197.51,Z 308.209,A -85,B 0,C 180,E1 -23092.429,E2 -23092.429} C_VEL
LIN {X 0,Y 195.298,Z 320.024,A -85,B 0,C 180,E1 -23093.452,E2 -23093.452} C_VEL
LIN {X 0,Y 193.625,Z 325.449,A -85,B 0,C 180,E1 -23093.941,E2 -23093.941} C_VEL
LIN {X 0,Y 189.151,Z 334.031,A -85,B 0,C 180,E1 -23094.599,E2 -23094.599} C_VEL
LIN {X 0,Y 184.321,Z 342.221,A -85,B 0,C 180,E1 -23095.472,E2 -23095.472} C_VEL
LIN {X 0,Y 182.121,Z 347.03,A -85,B 0,C 180,E1 -23096.3,E2 -23096.3} C_VEL
LIN {X 0,Y 178.578,Z 356.732,A -85,B 0,C 180,E1 -23098.57,E2 -23098.57} C_VEL
LIN {X 0,Y 175.055,Z 365.549,A -85,B 0,C 180,E1 -23101.199,E2 -23101.199} C_VEL
LIN {X 0,Y 171.941,Z 373.091,A -85,B 0,C 180,E1 -23104.059,E2 -23104.059} C_VEL
LIN {X 0,Y 168.868,Z 380.004,A -85,B 0,C 180,E1 -23107.358,E2 -23107.358} C_VEL
LIN {X 0,Y 166.672,Z 384.849,A -85,B 0,C 180,E1 -23110.286,E2 -23110.286} C_VEL
LIN {X 0,Y 164.484,Z 389.555,A -85,B 0,C 180,E1 -23113.875,E2 -23113.875} C_VEL
LIN {X 0,Y 163.098,Z 393.157,A -85,B 0,C 180,E1 -23117.558,E2 -23117.558} C_VEL
LIN {X 0,Y 162.41,Z 395.012,A -85,B 0,C 180,E1 -23120.032,E2 -23120.032} C_VEL
LIN {X 0,Y 161.763,Z 397.402,A -85,B 0,C 180,E1 -23125.015,E2 -23125.015} C_VEL
LIN {X 0,Y 161.762,Z 398.07,A -85,B 0,C 180,E1 -23127.818,E2 -23127.818} C_VEL
LIN {X 0,Y 161.833,Z 398.223,A -85,B 0,C 180,E1 -23130,E2 -23130} C_VEL
LIN {X 0,Y 161.76,Z 397.996,A -85,B 0,C 180,E1 -23132.49,E2 -23132.49} C_VEL
LIN {X 0,Y 161.999,Z 396.373,A -85,B 0,C 180,E1 -23137.478,E2 -23137.478} C_VEL
LIN {X 0,Y 162.41,Z 394.964,A -85,B 0,C 180,E1 -23139.968,E2 -23139.968} C_VEL
LIN {X 0,Y 163.483,Z 392.015,A -85,B 0,C 180,E1 -23143.677,E2 -23143.677} C_VEL
LIN {X 0,Y 165.111,Z 388.028,A -85,B 0,C 180,E1 -23147.335,E2 -23147.335} C_VEL
LIN {X 0,Y 167.957,Z 381.906,A -85,B 0,C 180,E1 -23151.477,E2 -23151.477} C_VEL
LIN {X 0,Y 171.248,Z 374.532,A -85,B 0,C 180,E1 -23155.238,E2 -23155.238} C_VEL
LIN {X 0,Y 174.383,Z 366.928,A -85,B 0,C 180,E1 -23158.265,E2 -23158.265} C_VEL
LIN {X 0,Y 177.821,Z 358.425,A -85,B 0,C 180,E1 -23160.917,E2 -23160.917} C_VEL
LIN {X 0,Y 181.652,Z 347.921,A -85,B 0,C 180,E1 -23163.458,E2 -23163.458} C_VEL
LIN {X 0,Y 185.421,Z 336.095,A -85,B 0,C 180,E1 -23165.645,E2 -23165.645} C_VEL
LIN {X 0,Y 188.533,Z 324.169,A -85,B 0,C 180,E1 -23167.283,E2 -23167.283} C_VEL
LIN {X 0,Y 191.153,Z 311.754,A -85,B 0,C 180,E1 -23168.516,E2 -23168.516} C_VEL
LIN {X 0,Y 193.193,Z 298.464,A -85,B 0,C 180,E1 -23169.408,E2 -23169.408} C_VEL
LIN {X 0,Y 194.374,Z 282.989,A -85,B 0,C 180,E1 -23170.033,E2 -23170.033} C_VEL
LIN {X 0,Y 196.297,Z 247.155,A -85,B 0,C 180,E1 -23171.248,E2 -23171.248} C_VEL
LIN {X 0,Y 195.732,Z 243.939,A -85,B 0,C 180,E1 -23171.546,E2 -23171.546} C_VEL
LIN {X 0,Y 190.759,Z 231.04,A -85,B 0,C 180,E1 -23173.526,E2 -23173.526} C_VEL
LIN {X 0,Y 184.889,Z 218.615,A -85,B 0,C 180,E1 -23175.941,E2 -23175.941} C_VEL
LIN {X 0,Y 179.468,Z 208.696,A -85,B 0,C 180,E1 -23178.327,E2 -23178.327} C_VEL
LIN {X 0,Y 174.518,Z 200.5,A -85,B 0,C 180,E1 -23180.692,E2 -23180.692} C_VEL
LIN {X 0,Y 171.369,Z 195.583,A -85,B 0,C 180,E1 -23182.315,E2 -23182.315} C_VEL
LIN {X 0,Y 168.882,Z 192.499,A -85,B 0,C 180,E1 -23183.629,E2 -23183.629} C_VEL
LIN {X 0,Y 168.002,Z 190.885,A -85,B 0,C 180,E1 -23184.15,E2 -23184.15} C_VEL
LIN {X 0,Y 165.574,Z 188.727,A -85,B 0,C 180,E1 -23185.483,E2 -23185.483} C_VEL
LIN {X 0,Y 164.446,Z 186.178,A -85,B 0,C 180,E1 -23186.249,E2 -23186.249} C_VEL
LIN {X 0,Y 164.339,Z 185.514,A -85,B 0,C 180,E1 -23186.4,E2 -23186.4} C_VEL
LIN {X 0,Y 164.37,Z 185.51,A -85,B 0,C 180,E1 -23189.13,E2 -23189.13} C_VEL
LIN {X 0,Y 164.395,Z 185.508,A -85,B 0,C 180,E1 -23194.691,E2 -23194.691} C_VEL
LIN {X 0,Y 164.485,Z 185.496,A -85,B 0,C 180,E1 -23200.051,E2 -23200.051} C_VEL
LIN {X 0,Y 164.524,Z 185.492,A -85,B 0,C 180,E1 -23205.149,E2 -23205.149} C_VEL
LIN {X 0,Y 164.769,Z 185.461,A -85,B 0,C 180,E1 -23210.177,E2 -23210.177} C_VEL
LIN {X 0,Y 164.832,Z 185.44,A -85,B 0,C 180,E1 -23212.651,E2 -23212.651} C_VEL
LIN {X 0,Y 165.049,Z 185.422,A -85,B 0,C 180,E1 -23217.56,E2 -23217.56} C_VEL
LIN {X 0,Y 165.294,Z 185.381,A -85,B 0,C 180,E1 -23220,E2 -23220} C_VEL
LIN {X 0,Y 164.763,Z 185.447,A -85,B 0,C 180,E1 -23224.894,E2 -23224.894} C_VEL
LIN {X 0,Y 164.831,Z 185.446,A -85,B 0,C 180,E1 -23227.349,E2 -23227.349} C_VEL
LIN {X 0,Y 164.704,Z 185.455,A -85,B 0,C 180,E1 -23231.062,E2 -23231.062} C_VEL
LIN {X 0,Y 164.498,Z 185.481,A -85,B 0,C 180,E1 -23237.402,E2 -23237.402} C_VEL
LIN {X 0,Y 164.476,Z 185.498,A -85,B 0,C 180,E1 -23239.989,E2 -23239.989} C_VEL
LIN {X 0,Y 164.395,Z 185.502,A -85,B 0,C 180,E1 -23246.134,E2 -23246.134} C_VEL
LIN {X 0,Y 164.377,Z 185.502,A -85,B 0,C 180,E1 -23251.228,E2 -23251.228} C_VEL
LIN {X 0,Y 164.353,Z 185.706,A -85,B 0,C 180,E1 -23254.033,E2 -23254.033} C_VEL
LIN {X 0,Y 165.281,Z 188.217,A -85,B 0,C 180,E1 -23254.699,E2 -23254.699} C_VEL
LIN {X 0,Y 167.362,Z 190.474,A -85,B 0,C 180,E1 -23255.884,E2 -23255.884} C_VEL
LIN {X 0,Y 168.242,Z 191.136,A -85,B 0,C 180,E1 -23256.346,E2 -23256.346} C_VEL
LIN {X 0,Y 170.28,Z 194.462,A -85,B 0,C 180,E1 -23257.502,E2 -23257.502} C_VEL
LIN {X 0,Y 172.043,Z 196.425,A -85,B 0,C 180,E1 -23258.395,E2 -23258.395} C_VEL
LIN {X 0,Y 174.797,Z 200.186,A -85,B 0,C 180,E1 -23259.766,E2 -23259.766} C_VEL
LIN {X 0,Y 180.876,Z 209.091,A -85,B 0,C 180,E1 -23262.557,E2 -23262.557} C_VEL
LIN {X 0,Y 187.283,Z 219.301,A -85,B 0,C 180,E1 -23265.209,E2 -23265.209} C_VEL
LIN {X 0,Y 190.594,Z 225.562,A -85,B 0,C 180,E1 -23266.515,E2 -23266.515} C_VEL
LIN {X 0,Y 196.481,Z 239.429,A -85,B 0,C 180,E1 -23268.797,E2 -23268.797} C_VEL
LIN {X 0,Y 196.699,Z 241.065,A -85,B 0,C 180,E1 -23268.931,E2 -23268.931} C_VEL
LIN {X 0,Y 193.999,Z 286.866,A -85,B 0,C 180,E1 -23270.481,E2 -23270.481} C_VEL
LIN {X 0,Y 192.341,Z 300.451,A -85,B 0,C 180,E1 -23271.287,E2 -23271.287} C_VEL
LIN {X 0,Y 190.168,Z 312.964,A -85,B 0,C 180,E1 -23272.426,E2 -23272.426} C_VEL
LIN {X 0,Y 187.587,Z 324.26,A -85,B 0,C 180,E1 -23273.838,E2 -23273.838} C_VEL
LIN {X 0,Y 184.228,Z 335.892,A -85,B 0,C 180,E1 -23275.758,E2 -23275.758} C_VEL
LIN {X 0,Y 180.722,Z 346.339,A -85,B 0,C 180,E1 -23278.004,E2 -23278.004} C_VEL
LIN {X 0,Y 177.592,Z 354.876,A -85,B 0,C 180,E1 -23280.353,E2 -23280.353} C_VEL
LIN {X 0,Y 174.506,Z 362.744,A -85,B 0,C 180,E1 -23283.063,E2 -23283.063} C_VEL
LIN {X 0,Y 171.016,Z 370.418,A -85,B 0,C 180,E1 -23286.379,E2 -23286.379} C_VEL
LIN {X 0,Y 167.634,Z 377.475,A -85,B 0,C 180,E1 -23290.403,E2 -23290.403} C_VEL
LIN {X 0,Y 165.446,Z 382.169,A -85,B 0,C 180,E1 -23293.972,E2 -23293.972} C_VEL
LIN {X 0,Y 163.807,Z 385.76,A -85,B 0,C 180,E1 -23297.613,E2 -23297.613} C_VEL
LIN {X 0,Y 163.051,Z 387.612,A -85,B 0,C 180,E1 -23300.072,E2 -23300.072} C_VEL
LIN {X 0,Y 162.479,Z 389.004,A -85,B 0,C 180,E1 -23302.544,E2 -23302.544} C_VEL
LIN {X 0,Y 161.926,Z 390.601,A -85,B 0,C 180,E1 -23307.512,E2 -23307.512} C_VEL
LIN {X 0,Y 161.887,Z 390.828,A -85,B 0,C 180,E1 -23310,E2 -23310} C_VEL
LIN {X 0,Y 162.029,Z 390.354,A -85,B 0,C 180,E1 -23313.945,E2 -23313.945} C_VEL
LIN {X 0,Y 162.472,Z 389.077,A -85,B 0,C 180,E1 -23317.456,E2 -23317.456} C_VEL
LIN {X 0,Y 163.002,Z 387.719,A -85,B 0,C 180,E1 -23319.931,E2 -23319.931} C_VEL
LIN {X 0,Y 164.26,Z 384.846,A -85,B 0,C 180,E1 -23323.61,E2 -23323.61} C_VEL
LIN {X 0,Y 166.108,Z 380.948,A -85,B 0,C 180,E1 -23327.227,E2 -23327.227} C_VEL
LIN {X 0,Y 168.487,Z 375.92,A -85,B 0,C 180,E1 -23330.766,E2 -23330.766} C_VEL
LIN {X 0,Y 171.515,Z 369.583,A -85,B 0,C 180,E1 -23334.19,E2 -23334.19} C_VEL
LIN {X 0,Y 174.777,Z 362.139,A -85,B 0,C 180,E1 -23337.333,E2 -23337.333} C_VEL
LIN {X 0,Y 178.083,Z 353.758,A -85,B 0,C 180,E1 -23340.145,E2 -23340.145} C_VEL
LIN {X 0,Y 181.804,Z 343.717,A -85,B 0,C 180,E1 -23342.765,E2 -23342.765} C_VEL
LIN {X 0,Y 185.383,Z 332.608,A -85,B 0,C 180,E1 -23344.987,E2 -23344.987} C_VEL
LIN {X 0,Y 188.368,Z 321.716,A -85,B 0,C 180,E1 -23346.652,E2 -23346.652} C_VEL
LIN {X 0,Y 190.966,Z 309.675,A -85,B 0,C 180,E1 -23348.056,E2 -23348.056} C_VEL
LIN {X 0,Y 192.957,Z 297.06,A -85,B 0,C 180,E1 -23349.111,E2 -23349.111} C_VEL
LIN {X 0,Y 194.351,Z 283.865,A -85,B 0,C 180,E1 -23349.788,E2 -23349.788} C_VEL
LIN {X 0,Y 196.842,Z 240.163,A -85,B 0,C 180,E1 -23351.257,E2 -23351.257} C_VEL
LIN {X 0,Y 191.095,Z 226.559,A -85,B 0,C 180,E1 -23353.482,E2 -23353.482} C_VEL
LIN {X 0,Y 187.952,Z 220.388,A -85,B 0,C 180,E1 -23354.727,E2 -23354.727} C_VEL
LIN {X 0,Y 182.268,Z 211.178,A -85,B 0,C 180,E1 -23357.055,E2 -23357.055} C_VEL
LIN {X 0,Y 177.097,Z 203.567,A -85,B 0,C 180,E1 -23359.357,E2 -23359.357} C_VEL
LIN {X 0,Y 174.246,Z 199.576,A -85,B 0,C 180,E1 -23360.721,E2 -23360.721} C_VEL
LIN {X 0,Y 171.326,Z 195.493,A -85,B 0,C 180,E1 -23362.211,E2 -23362.211} C_VEL
LIN {X 0,Y 168.854,Z 192.396,A -85,B 0,C 180,E1 -23363.529,E2 -23363.529} C_VEL
LIN {X 0,Y 168.095,Z 190.905,A -85,B 0,C 180,E1 -23363.988,E2 -23363.988} C_VEL
LIN {X 0,Y 165.708,Z 188.871,A -85,B 0,C 180,E1 -23365.298,E2 -23365.298} C_VEL
LIN {X 0,Y 164.498,Z 186.393,A -85,B 0,C 180,E1 -23366.105,E2 -23366.105} C_VEL
LIN {X 0,Y 164.344,Z 185.498,A -85,B 0,C 180,E1 -23366.312,E2 -23366.312} C_VEL
LIN {X 0,Y 164.406,Z 185.505,A -85,B 0,C 180,E1 -23369.138,E2 -23369.138} C_VEL
LIN {X 0,Y 164.417,Z 185.505,A -85,B 0,C 180,E1 -23374.694,E2 -23374.694} C_VEL
LIN {X 0,Y 164.485,Z 185.491,A -85,B 0,C 180,E1 -23380.051,E2 -23380.051} C_VEL
LIN {X 0,Y 164.536,Z 185.47,A -85,B 0,C 180,E1 -23385.15,E2 -23385.15} C_VEL
LIN {X 0,Y 164.798,Z 185.44,A -85,B 0,C 180,E1 -23390.178,E2 -23390.178} C_VEL
LIN {X 0,Y 164.846,Z 185.432,A -85,B 0,C 180,E1 -23392.652,E2 -23392.652} C_VEL
LIN {X 0,Y 165.05,Z 185.408,A -85,B 0,C 180,E1 -23397.559,E2 -23397.559} C_VEL
LIN {X 0,Y 165.294,Z 185.377,A -85,B 0,C 180,E1 -23400,E2 -23400} C_VEL
LIN {X 0,Y 164.77,Z 185.442,A -85,B 0,C 180,E1 -23404.894,E2 -23404.894} C_VEL
LIN {X 0,Y 164.851,Z 185.432,A -85,B 0,C 180,E1 -23407.348,E2 -23407.348} C_VEL
LIN {X 0,Y 164.742,Z 185.454,A -85,B 0,C 180,E1 -23411.131,E2 -23411.131} C_VEL
LIN {X 0,Y 164.503,Z 185.487,A -85,B 0,C 180,E1 -23417.401,E2 -23417.401} C_VEL
LIN {X 0,Y 164.473,Z 185.478,A -85,B 0,C 180,E1 -23419.989,E2 -23419.989} C_VEL
LIN {X 0,Y 164.385,Z 185.495,A -85,B 0,C 180,E1 -23426.128,E2 -23426.128} C_VEL
LIN {X 0,Y 164.378,Z 185.511,A -85,B 0,C 180,E1 -23432.374,E2 -23432.374} C_VEL
LIN {X 0,Y 164.339,Z 185.508,A -85,B 0,C 180,E1 -23433.426,E2 -23433.426} C_VEL
LIN {X 0,Y 165.291,Z 188.292,A -85,B 0,C 180,E1 -23434.172,E2 -23434.172} C_VEL
LIN {X 0,Y 167.573,Z 190.624,A -85,B 0,C 180,E1 -23435.467,E2 -23435.467} C_VEL
LIN {X 0,Y 168.416,Z 191.557,A -85,B 0,C 180,E1 -23435.932,E2 -23435.932} C_VEL
LIN {X 0,Y 170.467,Z 194.687,A -85,B 0,C 180,E1 -23437.082,E2 -23437.082} C_VEL
LIN {X 0,Y 172.396,Z 197.047,A -85,B 0,C 180,E1 -23438.074,E2 -23438.074} C_VEL
LIN {X 0,Y 178.549,Z 206.931,A -85,B 0,C 180,E1 -23441.111,E2 -23441.111} C_VEL
LIN {X 0,Y 185.105,Z 218.934,A -85,B 0,C 180,E1 -23444.033,E2 -23444.033} C_VEL
LIN {X 0,Y 191.209,Z 231.927,A -85,B 0,C 180,E1 -23446.546,E2 -23446.546} C_VEL
LIN {X 0,Y 196.156,Z 244.716,A -85,B 0,C 180,E1 -23448.508,E2 -23448.508} C_VEL
LIN {X 0,Y 196.412,Z 248.998,A -85,B 0,C 180,E1 -23448.777,E2 -23448.777} C_VEL
LIN {X 0,Y 193.685,Z 294.225,A -85,B 0,C 180,E1 -23450.308,E2 -23450.308} C_VEL
LIN {X 0,Y 192.028,Z 307.711,A -85,B 0,C 180,E1 -23451.121,E2 -23451.121} C_VEL
LIN {X 0,Y 189.554,Z 320.313,A -85,B 0,C 180,E1 -23452.221,E2 -23452.221} C_VEL
LIN {X 0,Y 186.783,Z 331.793,A -85,B 0,C 180,E1 -23453.657,E2 -23453.657} C_VEL
LIN {X 0,Y 183.375,Z 343.344,A -85,B 0,C 180,E1 -23455.577,E2 -23455.577} C_VEL
LIN {X 0,Y 182.121,Z 347.03,A -85,B 0,C 180,E1 -23456.3,E2 -23456.3} C_VEL
LIN {X 0,Y 179.854,Z 351.756,A -85,B 0,C 180,E1 -23457.214,E2 -23457.214} C_VEL
LIN {X 0,Y 174.56,Z 359.025,A -85,B 0,C 180,E1 -23458.601,E2 -23458.601} C_VEL
LIN {X 0,Y 169.262,Z 365.722,A -85,B 0,C 180,E1 -23460.249,E2 -23460.249} C_VEL
LIN {X 0,Y 167.033,Z 369.514,A -85,B 0,C 180,E1 -23461.552,E2 -23461.552} C_VEL
LIN {X 0,Y 164.002,Z 376.458,A -85,B 0,C 180,E1 -23464.626,E2 -23464.626} C_VEL
LIN {X 0,Y 160.914,Z 382.869,A -85,B 0,C 180,E1 -23468.208,E2 -23468.208} C_VEL
LIN {X 0,Y 158.335,Z 387.961,A -85,B 0,C 180,E1 -23471.898,E2 -23471.898} C_VEL
LIN {X 0,Y 156.556,Z 391.921,A -85,B 0,C 180,E1 -23475.706,E2 -23475.706} C_VEL
LIN {X 0,Y 155.413,Z 394.851,A -85,B 0,C 180,E1 -23479.579,E2 -23479.579} C_VEL
LIN {X 0,Y 154.691,Z 397.24,A -85,B 0,C 180,E1 -23484.787,E2 -23484.787} C_VEL
LIN {X 0,Y 154.663,Z 397.981,A -85,B 0,C 180,E1 -23488.592,E2 -23488.592} C_VEL
LIN {X 0,Y 154.676,Z 397.965,A -85,B 0,C 180,E1 -23491.596,E2 -23491.596} C_VEL
LIN {X 0,Y 154.699,Z 397.216,A -85,B 0,C 180,E1 -23495.213,E2 -23495.213} C_VEL
LIN {X 0,Y 154.949,Z 396.21,A -85,B 0,C 180,E1 -23497.821,E2 -23497.821} C_VEL
LIN {X 0,Y 155.413,Z 394.801,A -85,B 0,C 180,E1 -23500.421,E2 -23500.421} C_VEL
LIN {X 0,Y 156.556,Z 391.851,A -85,B 0,C 180,E1 -23504.294,E2 -23504.294} C_VEL
LIN {X 0,Y 158.335,Z 387.864,A -85,B 0,C 180,E1 -23508.102,E2 -23508.102} C_VEL
LIN {X 0,Y 161.313,Z 381.74,A -85,B 0,C 180,E1 -23512.409,E2 -23512.409} C_VEL
LIN {X 0,Y 164.566,Z 374.928,A -85,B 0,C 180,E1 -23516.03,E2 -23516.03} C_VEL
LIN {X 0,Y 168.139,Z 366.763,A -85,B 0,C 180,E1 -23519.415,E2 -23519.415} C_VEL
LIN {X 0,Y 171.767,Z 358.26,A -85,B 0,C 180,E1 -23522.134,E2 -23522.134} C_VEL
LIN {X 0,Y 175.774,Z 347.755,A -85,B 0,C 180,E1 -23524.733,E2 -23524.733} C_VEL
LIN {X 0,Y 179.699,Z 335.928,A -85,B 0,C 180,E1 -23526.964,E2 -23526.964} C_VEL
LIN {X 0,Y 182.944,Z 324.001,A -85,B 0,C 180,E1 -23528.628,E2 -23528.628} C_VEL
LIN {X 0,Y 185.668,Z 311.585,A -85,B 0,C 180,E1 -23529.876,E2 -23529.876} C_VEL
LIN {X 0,Y 187.727,Z 298.603,A -85,B 0,C 180,E1 -23530.767,E2 -23530.767} C_VEL
LIN {X 0,Y 188.888,Z 284.551,A -85,B 0,C 180,E1 -23531.359,E2 -23531.359} C_VEL
LIN {X 0,Y 190.958,Z 248.31,A -85,B 0,C 180,E1 -23532.602,E2 -23532.602} C_VEL
LIN {X 0,Y 189.664,Z 244.029,A -85,B 0,C 180,E1 -23533.176,E2 -23533.176} C_VEL
LIN {X 0,Y 185.022,Z 232.314,A -85,B 0,C 180,E1 -23535.158,E2 -23535.158} C_VEL
LIN {X 0,Y 179.461,Z 220.706,A -85,B 0,C 180,E1 -23537.629,E2 -23537.629} C_VEL
LIN {X 0,Y 173.9,Z 210.5,A -85,B 0,C 180,E1 -23540.304,E2 -23540.304} C_VEL
LIN {X 0,Y 168.574,Z 201.634,A -85,B 0,C 180,E1 -23543.133,E2 -23543.133} C_VEL
LIN {X 0,Y 165.807,Z 198.154,A -85,B 0,C 180,E1 -23544.672,E2 -23544.672} C_VEL
LIN {X 0,Y 164.767,Z 196.712,A -85,B 0,C 180,E1 -23545.289,E2 -23545.289} C_VEL
LIN {X 0,Y 162.317,Z 193.896,A -85,B 0,C 180,E1 -23546.771,E2 -23546.771} C_VEL
LIN {X 0,Y 161.209,Z 191.865,A -85,B 0,C 180,E1 -23547.536,E2 -23547.536} C_VEL
LIN {X 0,Y 158.762,Z 189.865,A -85,B 0,C 180,E1 -23549.113,E2 -23549.113} C_VEL
LIN {X 0,Y 157.539,Z 187.599,A -85,B 0,C 180,E1 -23550.06,E2 -23550.06} C_VEL
LIN {X 0,Y 157.25,Z 186.397,A -85,B 0,C 180,E1 -23550.369,E2 -23550.369} C_VEL
LIN {X 0,Y 157.309,Z 186.381,A -85,B 0,C 180,E1 -23553.464,E2 -23553.464} C_VEL
LIN {X 0,Y 157.393,Z 186.38,A -85,B 0,C 180,E1 -23559.669,E2 -23559.669} C_VEL
LIN {X 0,Y 157.454,Z 186.372,A -85,B 0,C 180,E1 -23564.466,E2 -23564.466} C_VEL
LIN {X 0,Y 157.69,Z 186.339,A -85,B 0,C 180,E1 -23569.731,E2 -23569.731} C_VEL
LIN {X 0,Y 157.768,Z 186.322,A -85,B 0,C 180,E1 -23572.32,E2 -23572.32} C_VEL
LIN {X 0,Y 158.257,Z 186.257,A -85,B 0,C 180,E1 -23580,E2 -23580} C_VEL
LIN {X 0,Y 157.768,Z 186.328,A -85,B 0,C 180,E1 -23587.68,E2 -23587.68} C_VEL
LIN {X 0,Y 157.638,Z 186.334,A -85,B 0,C 180,E1 -23591.237,E2 -23591.237} C_VEL
LIN {X 0,Y 157.461,Z 186.366,A -85,B 0,C 180,E1 -23595.534,E2 -23595.534} C_VEL
LIN {X 0,Y 157.372,Z 186.378,A -85,B 0,C 180,E1 -23600.933,E2 -23600.933} C_VEL
LIN {X 0,Y 157.315,Z 186.379,A -85,B 0,C 180,E1 -23606.685,E2 -23606.685} C_VEL
LIN {X 0,Y 157.327,Z 186.526,A -85,B 0,C 180,E1 -23610.077,E2 -23610.077} C_VEL
LIN {X 0,Y 158.277,Z 189.094,A -85,B 0,C 180,E1 -23610.894,E2 -23610.894} C_VEL
LIN {X 0,Y 160.111,Z 191.222,A -85,B 0,C 180,E1 -23612.159,E2 -23612.159} C_VEL
LIN {X 0,Y 161.53,Z 192.268,A -85,B 0,C 180,E1 -23613.04,E2 -23613.04} C_VEL
LIN {X 0,Y 163.436,Z 195.419,A -85,B 0,C 180,E1 -23614.303,E2 -23614.303} C_VEL
LIN {X 0,Y 165.591,Z 197.66,A -85,B 0,C 180,E1 -23615.553,E2 -23615.553} C_VEL
LIN {X 0,Y 168.043,Z 201.109,A -85,B 0,C 180,E1 -23616.956,E2 -23616.956} C_VEL
LIN {X 0,Y 172.564,Z 207.469,A -85,B 0,C 180,E1 -23619.333,E2 -23619.333} C_VEL
LIN {X 0,Y 177.45,Z 214.696,A -85,B 0,C 180,E1 -23621.667,E2 -23621.667} C_VEL
LIN {X 0,Y 183.493,Z 224.594,A -85,B 0,C 180,E1 -23624.306,E2 -23624.306} C_VEL
LIN {X 0,Y 186.717,Z 231.005,A -85,B 0,C 180,E1 -23625.657,E2 -23625.657} C_VEL
LIN {X 0,Y 191.348,Z 242.184,A -85,B 0,C 180,E1 -23627.566,E2 -23627.566} C_VEL
LIN {X 0,Y 188.592,Z 286.937,A -85,B 0,C 180,E1 -23629.105,E2 -23629.105} C_VEL
LIN {X 0,Y 186.909,Z 300.34,A -85,B 0,C 180,E1 -23629.906,E2 -23629.906} C_VEL
LIN {X 0,Y 184.604,Z 313.133,A -85,B 0,C 180,E1 -23631.085,E2 -23631.085} C_VEL
LIN {X 0,Y 181.903,Z 324.427,A -85,B 0,C 180,E1 -23632.518,E2 -23632.518} C_VEL
LIN {X 0,Y 178.421,Z 336.057,A -85,B 0,C 180,E1 -23634.479,E2 -23634.479} C_VEL
LIN {X 0,Y 174.723,Z 346.505,A -85,B 0,C 180,E1 -23636.767,E2 -23636.767} C_VEL
LIN {X 0,Y 170.958,Z 356.281,A -85,B 0,C 180,E1 -23639.575,E2 -23639.575} C_VEL
LIN {X 0,Y 167.534,Z 364.283,A -85,B 0,C 180,E1 -23642.52,E2 -23642.52} C_VEL
LIN {X 0,Y 164,Z 371.692,A -85,B 0,C 180,E1 -23645.977,E2 -23645.977} C_VEL
LIN {X 0,Y 160.948,Z 377.639,A -85,B 0,C 180,E1 -23649.554,E2 -23649.554} C_VEL
LIN {X 0,Y 158.622,Z 382.333,A -85,B 0,C 180,E1 -23653.262,E2 -23653.262} C_VEL
LIN {X 0,Y 156.874,Z 385.923,A -85,B 0,C 180,E1 -23657.056,E2 -23657.056} C_VEL
LIN {X 0,Y 156.055,Z 387.775,A -85,B 0,C 180,E1 -23659.622,E2 -23659.622} C_VEL
LIN {X 0,Y 155.436,Z 389.166,A -85,B 0,C 180,E1 -23662.204,E2 -23662.204} C_VEL
LIN {X 0,Y 154.87,Z 390.64,A -85,B 0,C 180,E1 -23666.726,E2 -23666.726} C_VEL
LIN {X 0,Y 154.794,Z 390.99,A -85,B 0,C 180,E1 -23670,E2 -23670} C_VEL
LIN {X 0,Y 154.869,Z 390.673,A -85,B 0,C 180,E1 -23673.269,E2 -23673.269} C_VEL
LIN {X 0,Y 155.429,Z 389.239,A -85,B 0,C 180,E1 -23677.796,E2 -23677.796} C_VEL
LIN {X 0,Y 156.017,Z 387.88,A -85,B 0,C 180,E1 -23680.38,E2 -23680.38} C_VEL
LIN {X 0,Y 157.368,Z 385.007,A -85,B 0,C 180,E1 -23684.219,E2 -23684.219} C_VEL
LIN {X 0,Y 159.344,Z 381.109,A -85,B 0,C 180,E1 -23687.983,E2 -23687.983} C_VEL
LIN {X 0,Y 161.848,Z 376.081,A -85,B 0,C 180,E1 -23691.66,E2 -23691.66} C_VEL
LIN {X 0,Y 165.076,Z 369.743,A -85,B 0,C 180,E1 -23695.197,E2 -23695.197} C_VEL
LIN {X 0,Y 168.37,Z 362.547,A -85,B 0,C 180,E1 -23698.352,E2 -23698.352} C_VEL
LIN {X 0,Y 172.046,Z 353.739,A -85,B 0,C 180,E1 -23701.388,E2 -23701.388} C_VEL
LIN {X 0,Y 175.861,Z 343.876,A -85,B 0,C 180,E1 -23704.02,E2 -23704.02} C_VEL
LIN {X 0,Y 179.616,Z 332.766,A -85,B 0,C 180,E1 -23706.285,E2 -23706.285} C_VEL
LIN {X 0,Y 182.737,Z 321.872,A -85,B 0,C 180,E1 -23707.977,E2 -23707.977} C_VEL
LIN {X 0,Y 185.434,Z 309.83,A -85,B 0,C 180,E1 -23709.407,E2 -23709.407} C_VEL
LIN {X 0,Y 187.44,Z 297.701,A -85,B 0,C 180,E1 -23710.446,E2 -23710.446} C_VEL
LIN {X 0,Y 188.942,Z 284.3,A -85,B 0,C 180,E1 -23711.151,E2 -23711.151} C_VEL
LIN {X 0,Y 191.389,Z 242.117,A -85,B 0,C 180,E1 -23712.615,E2 -23712.615} C_VEL
LIN {X 0,Y 185.605,Z 228.462,A -85,B 0,C 180,E1 -23715.017,E2 -23715.017} C_VEL
LIN {X 0,Y 181.062,Z 220.339,A -85,B 0,C 180,E1 -23716.943,E2 -23716.943} C_VEL
LIN {X 0,Y 174.217,Z 209.707,A -85,B 0,C 180,E1 -23720.089,E2 -23720.089} C_VEL
LIN {X 0,Y 168.242,Z 201.253,A -85,B 0,C 180,E1 -23723.188,E2 -23723.188} C_VEL
LIN {X 0,Y 165.604,Z 197.718,A -85,B 0,C 180,E1 -23724.692,E2 -23724.692} C_VEL
LIN {X 0,Y 164.517,Z 196.488,A -85,B 0,C 180,E1 -23725.326,E2 -23725.326} C_VEL
LIN {X 0,Y 162.115,Z 193.499,A -85,B 0,C 180,E1 -23726.816,E2 -23726.816} C_VEL
LIN {X 0,Y 161.328,Z 191.909,A -85,B 0,C 180,E1 -23727.377,E2 -23727.377} C_VEL
LIN {X 0,Y 158.905,Z 190.002,A -85,B 0,C 180,E1 -23728.94,E2 -23728.94} C_VEL
LIN {X 0,Y 157.574,Z 187.572,A -85,B 0,C 180,E1 -23729.975,E2 -23729.975} C_VEL
LIN {X 0,Y 157.304,Z 186.38,A -85,B 0,C 180,E1 -23730.38,E2 -23730.38} C_VEL
LIN {X 0,Y 157.322,Z 186.378,A -85,B 0,C 180,E1 -23733.466,E2 -23733.466} C_VEL
LIN {X 0,Y 157.394,Z 186.369,A -85,B 0,C 180,E1 -23739.667,E2 -23739.667} C_VEL
LIN {X 0,Y 157.462,Z 186.348,A -85,B 0,C 180,E1 -23744.466,E2 -23744.466} C_VEL
LIN {X 0,Y 157.726,Z 186.323,A -85,B 0,C 180,E1 -23749.733,E2 -23749.733} C_VEL
LIN {X 0,Y 157.785,Z 186.309,A -85,B 0,C 180,E1 -23752.321,E2 -23752.321} C_VEL
LIN {X 0,Y 158.257,Z 186.252,A -85,B 0,C 180,E1 -23760,E2 -23760} C_VEL
LIN {X 0,Y 157.808,Z 186.311,A -85,B 0,C 180,E1 -23767.678,E2 -23767.678} C_VEL
LIN {X 0,Y 157.673,Z 186.332,A -85,B 0,C 180,E1 -23771.303,E2 -23771.303} C_VEL
LIN {X 0,Y 157.471,Z 186.363,A -85,B 0,C 180,E1 -23775.532,E2 -23775.532} C_VEL
LIN {X 0,Y 157.367,Z 186.368,A -85,B 0,C 180,E1 -23780.933,E2 -23780.933} C_VEL
LIN {X 0,Y 157.309,Z 186.38,A -85,B 0,C 180,E1 -23786.681,E2 -23786.681} C_VEL
LIN {X 0,Y 157.278,Z 186.383,A -85,B 0,C 180,E1 -23789.442,E2 -23789.442} C_VEL
LIN {X 0,Y 158.097,Z 188.867,A -85,B 0,C 180,E1 -23790.191,E2 -23790.191} C_VEL
LIN {X 0,Y 160.332,Z 191.346,A -85,B 0,C 180,E1 -23791.736,E2 -23791.736} C_VEL
LIN {X 0,Y 161.522,Z 192.297,A -85,B 0,C 180,E1 -23792.486,E2 -23792.486} C_VEL
LIN {X 0,Y 163.485,Z 195.478,A -85,B 0,C 180,E1 -23793.791,E2 -23793.791} C_VEL
LIN {X 0,Y 165.476,Z 197.548,A -85,B 0,C 180,E1 -23794.956,E2 -23794.956} C_VEL
LIN {X 0,Y 168.114,Z 201.174,A -85,B 0,C 180,E1 -23796.471,E2 -23796.471} C_VEL
LIN {X 0,Y 169.73,Z 203.582,A -85,B 0,C 180,E1 -23797.364,E2 -23797.364} C_VEL
LIN {X 0,Y 174.845,Z 212.019,A -85,B 0,C 180,E1 -23800.026,E2 -23800.026} C_VEL
LIN {X 0,Y 181.092,Z 223.738,A -85,B 0,C 180,E1 -23802.984,E2 -23802.984} C_VEL
LIN {X 0,Y 186.685,Z 235.992,A -85,B 0,C 180,E1 -23805.437,E2 -23805.437} C_VEL
LIN {X 0,Y 191.028,Z 247.497,A -85,B 0,C 180,E1 -23807.278,E2 -23807.278} C_VEL
LIN {X 0,Y 190.411,Z 260.592,A -85,B 0,C 180,E1 -23807.763,E2 -23807.763} C_VEL
LIN {X 0,Y 188.239,Z 294.604,A -85,B 0,C 180,E1 -23808.959,E2 -23808.959} C_VEL
LIN {X 0,Y 186.422,Z 308.265,A -85,B 0,C 180,E1 -23809.8,E2 -23809.8} C_VEL
LIN {X 0,Y 183.914,Z 320.564,A -85,B 0,C 180,E1 -23810.912,E2 -23810.912} C_VEL
LIN {X 0,Y 180.659,Z 333.219,A -85,B 0,C 180,E1 -23812.566,E2 -23812.566} C_VEL
LIN {X 0,Y 177.136,Z 344.479,A -85,B 0,C 180,E1 -23814.532,E2 -23814.532} C_VEL
LIN {X 0,Y 173.308,Z 354.617,A -85,B 0,C 180,E1 -23816.808,E2 -23816.808} C_VEL
LIN {X 0,Y 169.543,Z 363.757,A -85,B 0,C 180,E1 -23819.483,E2 -23819.483} C_VEL
LIN {X 0,Y 167.033,Z 369.514,A -85,B 0,C 180,E1 -23821.552,E2 -23821.552} C_VEL
LIN {X 0,Y 164.841,Z 373.176,A -85,B 0,C 180,E1 -23822.961,E2 -23822.961} C_VEL
LIN {X 0,Y 159.66,Z 378.612,A -85,B 0,C 180,E1 -23825.245,E2 -23825.245} C_VEL
LIN {X 0,Y 154.547,Z 383.454,A -85,B 0,C 180,E1 -23827.816,E2 -23827.816} C_VEL
LIN {X 0,Y 152.522,Z 386.049,A -85,B 0,C 180,E1 -23829.644,E2 -23829.644} C_VEL
LIN {X 0,Y 150.176,Z 390.538,A -85,B 0,C 180,E1 -23833.693,E2 -23833.693} C_VEL
LIN {X 0,Y 149.172,Z 392.832,A -85,B 0,C 180,E1 -23836.375,E2 -23836.375} C_VEL
LIN {X 0,Y 148.401,Z 394.688,A -85,B 0,C 180,E1 -23839.081,E2 -23839.081} C_VEL
LIN {X 0,Y 147.619,Z 397.078,A -85,B 0,C 180,E1 -23844.536,E2 -23844.536} C_VEL
LIN {X 0,Y 147.606,Z 397.855,A -85,B 0,C 180,E1 -23849.11,E2 -23849.11} C_VEL
LIN {X 0,Y 147.568,Z 397.671,A -85,B 0,C 180,E1 -23852.73,E2 -23852.73} C_VEL
LIN {X 0,Y 147.626,Z 397.053,A -85,B 0,C 180,E1 -23855.464,E2 -23855.464} C_VEL
LIN {X 0,Y 147.899,Z 396.047,A -85,B 0,C 180,E1 -23858.196,E2 -23858.196} C_VEL
LIN {X 0,Y 148.401,Z 394.638,A -85,B 0,C 180,E1 -23860.92,E2 -23860.92} C_VEL
LIN {X 0,Y 149.655,Z 391.687,A -85,B 0,C 180,E1 -23864.969,E2 -23864.969} C_VEL
LIN {X 0,Y 151.594,Z 387.701,A -85,B 0,C 180,E1 -23868.937,E2 -23868.937} C_VEL
LIN {X 0,Y 154.731,Z 381.576,A -85,B 0,C 180,E1 -23873.418,E2 -23873.418} C_VEL
LIN {X 0,Y 157.545,Z 376.128,A -85,B 0,C 180,E1 -23876.493,E2 -23876.493} C_VEL
LIN {X 0,Y 161.269,Z 368.088,A -85,B 0,C 180,E1 -23880.077,E2 -23880.077} C_VEL
LIN {X 0,Y 164.976,Z 359.898,A -85,B 0,C 180,E1 -23882.898,E2 -23882.898} C_VEL
LIN {X 0,Y 169.115,Z 349.913,A -85,B 0,C 180,E1 -23885.578,E2 -23885.578} C_VEL
LIN {X 0,Y 173.152,Z 338.62,A -85,B 0,C 180,E1 -23887.872,E2 -23887.872} C_VEL
LIN {X 0,Y 176.464,Z 327.553,A -85,B 0,C 180,E1 -23889.585,E2 -23889.585} C_VEL
LIN {X 0,Y 179.49,Z 315.269,A -85,B 0,C 180,E1 -23890.984,E2 -23890.984} C_VEL
LIN {X 0,Y 181.906,Z 301.929,A -85,B 0,C 180,E1 -23892.015,E2 -23892.015} C_VEL
LIN {X 0,Y 183.392,Z 288.051,A -85,B 0,C 180,E1 -23892.693,E2 -23892.693} C_VEL
LIN {X 0,Y 185.695,Z 249.891,A -85,B 0,C 180,E1 -23894.02,E2 -23894.02} C_VEL
LIN {X 0,Y 181.28,Z 237.969,A -85,B 0,C 180,E1 -23896.036,E2 -23896.036} C_VEL
LIN {X 0,Y 176.034,Z 226.488,A -85,B 0,C 180,E1 -23898.51,E2 -23898.51} C_VEL
LIN {X 0,Y 170.633,Z 216.11,A -85,B 0,C 180,E1 -23901.266,E2 -23901.266} C_VEL
LIN {X 0,Y 165.351,Z 207.24,A -85,B 0,C 180,E1 -23904.23,E2 -23904.23} C_VEL
LIN {X 0,Y 162.462,Z 203.231,A -85,B 0,C 180,E1 -23905.967,E2 -23905.967} C_VEL
LIN {X 0,Y 159.465,Z 199.583,A -85,B 0,C 180,E1 -23907.885,E2 -23907.885} C_VEL
LIN {X 0,Y 158.488,Z 198.066,A -85,B 0,C 180,E1 -23908.576,E2 -23908.576} C_VEL
LIN {X 0,Y 155.934,Z 195.454,A -85,B 0,C 180,E1 -23910.372,E2 -23910.372} C_VEL
LIN {X 0,Y 154.59,Z 192.977,A -85,B 0,C 180,E1 -23911.487,E2 -23911.487} C_VEL
LIN {X 0,Y 152.057,Z 191.16,A -85,B 0,C 180,E1 -23913.469,E2 -23913.469} C_VEL
LIN {X 0,Y 150.605,Z 188.847,A -85,B 0,C 180,E1 -23914.84,E2 -23914.84} C_VEL
LIN {X 0,Y 150.223,Z 187.271,A -85,B 0,C 180,E1 -23915.376,E2 -23915.376} C_VEL
LIN {X 0,Y 150.36,Z 187.247,A -85,B 0,C 180,E1 -23920.902,E2 -23920.902} C_VEL
LIN {X 0,Y 150.436,Z 187.235,A -85,B 0,C 180,E1 -23926.492,E2 -23926.492} C_VEL
LIN {X 0,Y 150.612,Z 187.216,A -85,B 0,C 180,E1 -23929.243,E2 -23929.243} C_VEL
LIN {X 0,Y 150.706,Z 187.203,A -85,B 0,C 180,E1 -23931.958,E2 -23931.958} C_VEL
LIN {X 0,Y 151.217,Z 187.133,A -85,B 0,C 180,E1 -23940,E2 -23940} C_VEL
LIN {X 0,Y 150.705,Z 187.211,A -85,B 0,C 180,E1 -23948.042,E2 -23948.042} C_VEL
LIN {X 0,Y 150.578,Z 187.212,A -85,B 0,C 180,E1 -23951.438,E2 -23951.438} C_VEL
LIN {X 0,Y 150.369,Z 187.243,A -85,B 0,C 180,E1 -23956.286,E2 -23956.286} C_VEL
LIN {X 0,Y 150.353,Z 187.253,A -85,B 0,C 180,E1 -23960.794,E2 -23960.794} C_VEL
LIN {X 0,Y 150.264,Z 187.406,A -85,B 0,C 180,E1 -23965.091,E2 -23965.091} C_VEL
LIN {X 0,Y 151.013,Z 189.684,A -85,B 0,C 180,E1 -23965.942,E2 -23965.942} C_VEL
LIN {X 0,Y 153.035,Z 192.091,A -85,B 0,C 180,E1 -23967.709,E2 -23967.709} C_VEL
LIN {X 0,Y 154.875,Z 193.333,A -85,B 0,C 180,E1 -23969.105,E2 -23969.105} C_VEL
LIN {X 0,Y 156.67,Z 196.412,A -85,B 0,C 180,E1 -23970.546,E2 -23970.546} C_VEL
LIN {X 0,Y 158.986,Z 198.666,A -85,B 0,C 180,E1 -23972.131,E2 -23972.131} C_VEL
LIN {X 0,Y 161.474,Z 202.209,A -85,B 0,C 180,E1 -23973.8,E2 -23973.8} C_VEL
LIN {X 0,Y 162.912,Z 203.904,A -85,B 0,C 180,E1 -23974.683,E2 -23974.683} C_VEL
LIN {X 0,Y 166.486,Z 208.947,A -85,B 0,C 180,E1 -23976.792,E2 -23976.792} C_VEL
LIN {X 0,Y 171.46,Z 216.183,A -85,B 0,C 180,E1 -23979.446,E2 -23979.446} C_VEL
LIN {X 0,Y 178.08,Z 226.918,A -85,B 0,C 180,E1 -23982.616,E2 -23982.616} C_VEL
LIN {X 0,Y 181.683,Z 233.72,A -85,B 0,C 180,E1 -23984.225,E2 -23984.225} C_VEL
LIN {X 0,Y 186.051,Z 244.379,A -85,B 0,C 180,E1 -23986.162,E2 -23986.162} C_VEL
LIN {X 0,Y 183.362,Z 286.407,A -85,B 0,C 180,E1 -23987.624,E2 -23987.624} C_VEL
LIN {X 0,Y 181.749,Z 299.45,A -85,B 0,C 180,E1 -23988.394,E2 -23988.394} C_VEL
LIN {X 0,Y 179.836,Z 309.919,A -85,B 0,C 180,E1 -23989.296,E2 -23989.296} C_VEL
LIN {X 0,Y 176.796,Z 322.865,A -85,B 0,C 180,E1 -23990.871,E2 -23990.871} C_VEL
LIN {X 0,Y 173.578,Z 333.598,A -85,B 0,C 180,E1 -23992.603,E2 -23992.603} C_VEL
LIN {X 0,Y 169.662,Z 344.538,A -85,B 0,C 180,E1 -23994.918,E2 -23994.918} C_VEL
LIN {X 0,Y 166.088,Z 353.431,A -85,B 0,C 180,E1 -23997.35,E2 -23997.35} C_VEL
LIN {X 0,Y 162.301,Z 362.159,A -85,B 0,C 180,E1 -24000.411,E2 -24000.411} C_VEL
LIN {X 0,Y 158.711,Z 369.579,A -85,B 0,C 180,E1 -24003.716,E2 -24003.716} C_VEL
LIN {X 0,Y 155.341,Z 375.993,A -85,B 0,C 180,E1 -24007.383,E2 -24007.383} C_VEL
LIN {X 0,Y 152.623,Z 381.079,A -85,B 0,C 180,E1 -24011.196,E2 -24011.196} C_VEL
LIN {X 0,Y 150.528,Z 385.026,A -85,B 0,C 180,E1 -24015.12,E2 -24015.12} C_VEL
LIN {X 0,Y 149.084,Z 387.938,A -85,B 0,C 180,E1 -24019.131,E2 -24019.131} C_VEL
LIN {X 0,Y 148.002,Z 390.318,A -85,B 0,C 180,E1 -24024.55,E2 -24024.55} C_VEL
LIN {X 0,Y 147.756,Z 390.925,A -85,B 0,C 180,E1 -24027.274,E2 -24027.274} C_VEL
LIN {X 0,Y 147.718,Z 391.151,A -85,B 0,C 180,E1 -24030,E2 -24030} C_VEL
LIN {X 0,Y 147.756,Z 390.956,A -85,B 0,C 180,E1 -24032.726,E2 -24032.726} C_VEL
LIN {X 0,Y 148.001,Z 390.369,A -85,B 0,C 180,E1 -24035.45,E2 -24035.45} C_VEL
LIN {X 0,Y 149.031,Z 388.042,A -85,B 0,C 180,E1 -24040.873,E2 -24040.873} C_VEL
LIN {X 0,Y 150.485,Z 385.169,A -85,B 0,C 180,E1 -24044.884,E2 -24044.884} C_VEL
LIN {X 0,Y 152.59,Z 381.271,A -85,B 0,C 180,E1 -24048.808,E2 -24048.808} C_VEL
LIN {X 0,Y 155.259,Z 376.242,A -85,B 0,C 180,E1 -24052.629,E2 -24052.629} C_VEL
LIN {X 0,Y 158.678,Z 369.903,A -85,B 0,C 180,E1 -24056.289,E2 -24056.289} C_VEL
LIN {X 0,Y 162.68,Z 361.486,A -85,B 0,C 180,E1 -24060.027,E2 -24060.027} C_VEL
LIN {X 0,Y 166.803,Z 352.12,A -85,B 0,C 180,E1 -24063.211,E2 -24063.211} C_VEL
LIN {X 0,Y 170.876,Z 341.761,A -85,B 0,C 180,E1 -24065.88,E2 -24065.88} C_VEL
LIN {X 0,Y 174.869,Z 330.076,A -85,B 0,C 180,E1 -24068.164,E2 -24068.164} C_VEL
LIN {X 0,Y 178.128,Z 318.41,A -85,B 0,C 180,E1 -24069.876,E2 -24069.876} C_VEL
LIN {X 0,Y 180.677,Z 306.273,A -85,B 0,C 180,E1 -24071.211,E2 -24071.211} C_VEL
LIN {X 0,Y 182.761,Z 293.391,A -85,B 0,C 180,E1 -24072.162,E2 -24072.162} C_VEL
LIN {X 0,Y 183.986,Z 280.488,A -85,B 0,C 180,E1 -24072.748,E2 -24072.748} C_VEL
LIN {X 0,Y 186.171,Z 244.407,A -85,B 0,C 180,E1 -24073.997,E2 -24073.997} C_VEL
LIN {X 0,Y 180.613,Z 231.208,A -85,B 0,C 180,E1 -24076.477,E2 -24076.477} C_VEL
LIN {X 0,Y 174.334,Z 220.636,A -85,B 0,C 180,E1 -24079.359,E2 -24079.359} C_VEL
LIN {X 0,Y 169.446,Z 213.158,A -85,B 0,C 180,E1 -24081.836,E2 -24081.836} C_VEL
LIN {X 0,Y 165.198,Z 207,A -85,B 0,C 180,E1 -24084.208,E2 -24084.208} C_VEL
LIN {X 0,Y 161.909,Z 202.58,A -85,B 0,C 180,E1 -24086.21,E2 -24086.21} C_VEL
LIN {X 0,Y 159.388,Z 199.394,A -85,B 0,C 180,E1 -24087.861,E2 -24087.861} C_VEL
LIN {X 0,Y 158.429,Z 197.973,A -85,B 0,C 180,E1 -24088.542,E2 -24088.542} C_VEL
LIN {X 0,Y 155.976,Z 195.423,A -85,B 0,C 180,E1 -24090.288,E2 -24090.288} C_VEL
LIN {X 0,Y 154.539,Z 192.941,A -85,B 0,C 180,E1 -24091.477,E2 -24091.477} C_VEL
LIN {X 0,Y 152.041,Z 191.123,A -85,B 0,C 180,E1 -24093.46,E2 -24093.46} C_VEL
LIN {X 0,Y 150.603,Z 188.816,A -85,B 0,C 180,E1 -24094.838,E2 -24094.838} C_VEL
LIN {X 0,Y 150.239,Z 187.269,A -85,B 0,C 180,E1 -24095.378,E2 -24095.378} C_VEL
LIN {X 0,Y 150.361,Z 187.256,A -85,B 0,C 180,E1 -24100.902,E2 -24100.902} C_VEL
LIN {X 0,Y 150.451,Z 187.233,A -85,B 0,C 180,E1 -24106.493,E2 -24106.493} C_VEL
LIN {X 0,Y 150.653,Z 187.209,A -85,B 0,C 180,E1 -24109.245,E2 -24109.245} C_VEL
LIN {X 0,Y 150.724,Z 187.186,A -85,B 0,C 180,E1 -24111.959,E2 -24111.959} C_VEL
LIN {X 0,Y 151.217,Z 187.128,A -85,B 0,C 180,E1 -24120,E2 -24120} C_VEL
LIN {X 0,Y 150.742,Z 187.193,A -85,B 0,C 180,E1 -24128.04,E2 -24128.04} C_VEL
LIN {X 0,Y 150.607,Z 187.209,A -85,B 0,C 180,E1 -24131.492,E2 -24131.492} C_VEL
LIN {X 0,Y 150.378,Z 187.252,A -85,B 0,C 180,E1 -24136.285,E2 -24136.285} C_VEL
LIN {X 0,Y 150.349,Z 187.24,A -85,B 0,C 180,E1 -24140.79,E2 -24140.79} C_VEL
LIN {X 0,Y 150.257,Z 187.327,A -85,B 0,C 180,E1 -24144.434,E2 -24144.434} C_VEL
LIN {X 0,Y 150.985,Z 189.684,A -85,B 0,C 180,E1 -24145.289,E2 -24145.289} C_VEL
LIN {X 0,Y 153.061,Z 192.068,A -85,B 0,C 180,E1 -24147.118,E2 -24147.118} C_VEL
LIN {X 0,Y 154.814,Z 193.288,A -85,B 0,C 180,E1 -24148.468,E2 -24148.468} C_VEL
LIN {X 0,Y 156.547,Z 196.228,A -85,B 0,C 180,E1 -24149.875,E2 -24149.875} C_VEL
LIN {X 0,Y 159.011,Z 198.687,A -85,B 0,C 180,E1 -24151.585,E2 -24151.585} C_VEL
LIN {X 0,Y 161.244,Z 201.936,A -85,B 0,C 180,E1 -24153.106,E2 -24153.106} C_VEL
LIN {X 0,Y 162.876,Z 203.875,A -85,B 0,C 180,E1 -24154.121,E2 -24154.121} C_VEL
LIN {X 0,Y 166.276,Z 208.661,A -85,B 0,C 180,E1 -24156.149,E2 -24156.149} C_VEL
LIN {X 0,Y 171.397,Z 217.398,A -85,B 0,C 180,E1 -24158.991,E2 -24158.991} C_VEL
LIN {X 0,Y 176.955,Z 228.18,A -85,B 0,C 180,E1 -24161.799,E2 -24161.799} C_VEL
LIN {X 0,Y 182.08,Z 239.717,A -85,B 0,C 180,E1 -24164.206,E2 -24164.206} C_VEL
LIN {X 0,Y 185.864,Z 249.926,A -85,B 0,C 180,E1 -24165.926,E2 -24165.926} C_VEL
LIN {X 0,Y 183.019,Z 293.701,A -85,B 0,C 180,E1 -24167.459,E2 -24167.459} C_VEL
LIN {X 0,Y 181.219,Z 307.367,A -85,B 0,C 180,E1 -24168.304,E2 -24168.304} C_VEL
LIN {X 0,Y 178.713,Z 319.306,A -85,B 0,C 180,E1 -24169.358,E2 -24169.358} C_VEL
LIN {X 0,Y 175.542,Z 331.478,A -85,B 0,C 180,E1 -24170.908,E2 -24170.908} C_VEL
LIN {X 0,Y 171.851,Z 343.027,A -85,B 0,C 180,E1 -24172.9,E2 -24172.9} C_VEL
LIN {X 0,Y 167.843,Z 353.426,A -85,B 0,C 180,E1 -24175.214,E2 -24175.214} C_VEL
LIN {X 0,Y 164.214,Z 361.931,A -85,B 0,C 180,E1 -24177.658,E2 -24177.658} C_VEL
LIN {X 0,Y 160.528,Z 369.943,A -85,B 0,C 180,E1 -24180.579,E2 -24180.579} C_VEL
LIN {X 0,Y 157.032,Z 377.451,A -85,B 0,C 180,E1 -24184.128,E2 -24184.128} C_VEL
LIN {X 0,Y 154.286,Z 382.707,A -85,B 0,C 180,E1 -24187.221,E2 -24187.221} C_VEL
LIN {X 0,Y 152.522,Z 386.049,A -85,B 0,C 180,E1 -24189.644,E2 -24189.644} C_VEL
LIN {X 0,Y 150.626,Z 388.448,A -85,B 0,C 180,E1 -24191.558,E2 -24191.558} C_VEL
LIN {X 0,Y 146.167,Z 391.731,A -85,B 0,C 180,E1 -24194.736,E2 -24194.736} C_VEL
LIN {X 0,Y 142.795,Z 393.829,A -85,B 0,C 180,E1 -24197.472,E2 -24197.472} C_VEL
LIN {X 0,Y 141.209,Z 395.136,A -85,B 0,C 180,E1 -24199.714,E2 -24199.714} C_VEL
LIN {X 0,Y 140.977,Z 395.483,A -85,B 0,C 180,E1 -24200.494,E2 -24200.494} C_VEL
LIN {X 0,Y 140.543,Z 396.916,A -85,B 0,C 180,E1 -24204.26,E2 -24204.26} C_VEL
LIN {X 0,Y 140.486,Z 397.525,A -85,B 0,C 180,E1 -24207.133,E2 -24207.133} C_VEL
LIN {X 0,Y 140.56,Z 397.737,A -85,B 0,C 180,E1 -24210,E2 -24210} C_VEL
LIN {X 0,Y 140.486,Z 397.509,A -85,B 0,C 180,E1 -24212.868,E2 -24212.868} C_VEL
LIN {X 0,Y 140.549,Z 396.89,A -85,B 0,C 180,E1 -24215.74,E2 -24215.74} C_VEL
LIN {X 0,Y 140.851,Z 395.884,A -85,B 0,C 180,E1 -24218.609,E2 -24218.609} C_VEL
LIN {X 0,Y 141.413,Z 394.474,A -85,B 0,C 180,E1 -24221.467,E2 -24221.467} C_VEL
LIN {X 0,Y 142.783,Z 391.524,A -85,B 0,C 180,E1 -24225.707,E2 -24225.707} C_VEL
LIN {X 0,Y 144.889,Z 387.537,A -85,B 0,C 180,E1 -24229.849,E2 -24229.849} C_VEL
LIN {X 0,Y 148.218,Z 381.411,A -85,B 0,C 180,E1 -24234.513,E2 -24234.513} C_VEL
LIN {X 0,Y 151.153,Z 375.962,A -85,B 0,C 180,E1 -24237.708,E2 -24237.708} C_VEL
LIN {X 0,Y 155.142,Z 367.923,A -85,B 0,C 180,E1 -24241.396,E2 -24241.396} C_VEL
LIN {X 0,Y 159.063,Z 359.734,A -85,B 0,C 180,E1 -24244.287,E2 -24244.287} C_VEL
LIN {X 0,Y 163.387,Z 349.747,A -85,B 0,C 180,E1 -24247.028,E2 -24247.028} C_VEL
LIN {X 0,Y 167.59,Z 338.453,A -85,B 0,C 180,E1 -24249.366,E2 -24249.366} C_VEL
LIN {X 0,Y 171.064,Z 327.386,A -85,B 0,C 180,E1 -24251.098,E2 -24251.098} C_VEL
LIN {X 0,Y 174.2,Z 315.1,A -85,B 0,C 180,E1 -24252.514,E2 -24252.514} C_VEL
LIN {X 0,Y 176.589,Z 302.446,A -85,B 0,C 180,E1 -24253.514,E2 -24253.514} C_VEL
LIN {X 0,Y 178.16,Z 288.987,A -85,B 0,C 180,E1 -24254.192,E2 -24254.192} C_VEL
LIN {X 0,Y 180.519,Z 251.856,A -85,B 0,C 180,E1 -24255.51,E2 -24255.51} C_VEL
LIN {X 0,Y 176.36,Z 240.672,A -85,B 0,C 180,E1 -24257.549,E2 -24257.549} C_VEL
LIN {X 0,Y 170.909,Z 228.607,A -85,B 0,C 180,E1 -24260.342,E2 -24260.342} C_VEL
LIN {X 0,Y 164.927,Z 217.262,A -85,B 0,C 180,E1 -24263.709,E2 -24263.709} C_VEL
LIN {X 0,Y 162.007,Z 212.57,A -85,B 0,C 180,E1 -24265.486,E2 -24265.486} C_VEL
LIN {X 0,Y 158.805,Z 208.211,A -85,B 0,C 180,E1 -24267.548,E2 -24267.548} C_VEL
LIN {X 0,Y 155.81,Z 204.136,A -85,B 0,C 180,E1 -24269.67,E2 -24269.67} C_VEL
LIN {X 0,Y 153.085,Z 200.833,A -85,B 0,C 180,E1 -24271.766,E2 -24271.766} C_VEL
LIN {X 0,Y 152.232,Z 199.412,A -85,B 0,C 180,E1 -24272.506,E2 -24272.506} C_VEL
LIN {X 0,Y 149.508,Z 196.921,A -85,B 0,C 180,E1 -24274.84,E2 -24274.84} C_VEL
LIN {X 0,Y 147.89,Z 193.946,A -85,B 0,C 180,E1 -24276.547,E2 -24276.547} C_VEL
LIN {X 0,Y 145.452,Z 192.412,A -85,B 0,C 180,E1 -24279.054,E2 -24279.054} C_VEL
LIN {X 0,Y 143.796,Z 189.948,A -85,B 0,C 180,E1 -24281.2,E2 -24281.2} C_VEL
LIN {X 0,Y 143.287,Z 188.122,A -85,B 0,C 180,E1 -24282.148,E2 -24282.148} C_VEL
LIN {X 0,Y 143.538,Z 188.092,A -85,B 0,C 180,E1 -24288.706,E2 -24288.706} C_VEL
LIN {X 0,Y 143.627,Z 188.088,A -85,B 0,C 180,E1 -24291.559,E2 -24291.559} C_VEL
LIN {X 0,Y 144.176,Z 188.009,A -85,B 0,C 180,E1 -24300,E2 -24300} C_VEL
LIN {X 0,Y 143.627,Z 188.095,A -85,B 0,C 180,E1 -24308.442,E2 -24308.442} C_VEL
LIN {X 0,Y 143.506,Z 188.092,A -85,B 0,C 180,E1 -24311.631,E2 -24311.631} C_VEL
LIN {X 0,Y 143.311,Z 188.134,A -85,B 0,C 180,E1 -24318.311,E2 -24318.311} C_VEL
LIN {X 0,Y 143.969,Z 190.339,A -85,B 0,C 180,E1 -24319.424,E2 -24319.424} C_VEL
LIN {X 0,Y 145.972,Z 192.903,A -85,B 0,C 180,E1 -24321.899,E2 -24321.899} C_VEL
LIN {X 0,Y 148.125,Z 194.268,A -85,B 0,C 180,E1 -24324.063,E2 -24324.063} C_VEL
LIN {X 0,Y 149.891,Z 197.389,A -85,B 0,C 180,E1 -24325.885,E2 -24325.885} C_VEL
LIN {X 0,Y 152.602,Z 199.856,A -85,B 0,C 180,E1 -24328.168,E2 -24328.168} C_VEL
LIN {X 0,Y 155.015,Z 203.401,A -85,B 0,C 180,E1 -24330.127,E2 -24330.127} C_VEL
LIN {X 0,Y 156.599,Z 205.107,A -85,B 0,C 180,E1 -24331.267,E2 -24331.267} C_VEL
LIN {X 0,Y 159.515,Z 208.951,A -85,B 0,C 180,E1 -24333.275,E2 -24333.275} C_VEL
LIN {X 0,Y 165.394,Z 217.385,A -85,B 0,C 180,E1 -24336.885,E2 -24336.885} C_VEL
LIN {X 0,Y 172.155,Z 228.201,A -85,B 0,C 180,E1 -24340.493,E2 -24340.493} C_VEL
LIN {X 0,Y 177.011,Z 237.122,A -85,B 0,C 180,E1 -24342.838,E2 -24342.838} C_VEL
LIN {X 0,Y 180.828,Z 246.565,A -85,B 0,C 180,E1 -24344.662,E2 -24344.662} C_VEL
LIN {X 0,Y 178.227,Z 286.205,A -85,B 0,C 180,E1 -24346.074,E2 -24346.074} C_VEL
LIN {X 0,Y 176.607,Z 299.135,A -85,B 0,C 180,E1 -24346.832,E2 -24346.832} C_VEL
LIN {X 0,Y 174.765,Z 308.943,A -85,B 0,C 180,E1 -24347.656,E2 -24347.656} C_VEL
LIN {X 0,Y 171.837,Z 321.269,A -85,B 0,C 180,E1 -24349.127,E2 -24349.127} C_VEL
LIN {X 0,Y 168.013,Z 333.765,A -85,B 0,C 180,E1 -24351.138,E2 -24351.138} C_VEL
LIN {X 0,Y 163.917,Z 344.703,A -85,B 0,C 180,E1 -24353.495,E2 -24353.495} C_VEL
LIN {X 0,Y 160.153,Z 353.594,A -85,B 0,C 180,E1 -24355.978,E2 -24355.978} C_VEL
LIN {X 0,Y 155.93,Z 362.797,A -85,B 0,C 180,E1 -24359.313,E2 -24359.313} C_VEL
LIN {X 0,Y 152.369,Z 369.743,A -85,B 0,C 180,E1 -24362.532,E2 -24362.532} C_VEL
LIN {X 0,Y 148.785,Z 376.158,A -85,B 0,C 180,E1 -24366.328,E2 -24366.328} C_VEL
LIN {X 0,Y 145.912,Z 381.242,A -85,B 0,C 180,E1 -24370.296,E2 -24370.296} C_VEL
LIN {X 0,Y 143.669,Z 385.189,A -85,B 0,C 180,E1 -24374.392,E2 -24374.392} C_VEL
LIN {X 0,Y 142.114,Z 388.101,A -85,B 0,C 180,E1 -24378.591,E2 -24378.591} C_VEL
LIN {X 0,Y 141.381,Z 389.492,A -85,B 0,C 180,E1 -24381.423,E2 -24381.423} C_VEL
LIN {X 0,Y 140.941,Z 390.48,A -85,B 0,C 180,E1 -24384.276,E2 -24384.276} C_VEL
LIN {X 0,Y 140.597,Z 391.245,A -85,B 0,C 180,E1 -24388.702,E2 -24388.702} C_VEL
LIN {X 0,Y 140.678,Z 391.118,A -85,B 0,C 180,E1 -24392.863,E2 -24392.863} C_VEL
LIN {X 0,Y 140.94,Z 390.531,A -85,B 0,C 180,E1 -24395.723,E2 -24395.723} C_VEL
LIN {X 0,Y 142.053,Z 388.204,A -85,B 0,C 180,E1 -24401.414,E2 -24401.414} C_VEL
LIN {X 0,Y 143.617,Z 385.331,A -85,B 0,C 180,E1 -24405.613,E2 -24405.613} C_VEL
LIN {X 0,Y 145.878,Z 381.432,A -85,B 0,C 180,E1 -24409.709,E2 -24409.709} C_VEL
LIN {X 0,Y 148.723,Z 376.403,A -85,B 0,C 180,E1 -24413.683,E2 -24413.683} C_VEL
LIN {X 0,Y 152.335,Z 370.064,A -85,B 0,C 180,E1 -24417.474,E2 -24417.474} C_VEL
LIN {X 0,Y 156.315,Z 362.164,A -85,B 0,C 180,E1 -24421.121,E2 -24421.121} C_VEL
LIN {X 0,Y 160.095,Z 354.058,A -85,B 0,C 180,E1 -24424.035,E2 -24424.035} C_VEL
LIN {X 0,Y 164.28,Z 344.194,A -85,B 0,C 180,E1 -24426.793,E2 -24426.793} C_VEL
LIN {X 0,Y 168.398,Z 333.08,A -85,B 0,C 180,E1 -24429.141,E2 -24429.141} C_VEL
LIN {X 0,Y 171.794,Z 322.184,A -85,B 0,C 180,E1 -24430.885,E2 -24430.885} C_VEL
LIN {X 0,Y 174.699,Z 310.139,A -85,B 0,C 180,E1 -24432.364,E2 -24432.364} C_VEL
LIN {X 0,Y 176.888,Z 298.006,A -85,B 0,C 180,E1 -24433.427,E2 -24433.427} C_VEL
LIN {X 0,Y 178.552,Z 284.327,A -85,B 0,C 180,E1 -24434.15,E2 -24434.15} C_VEL
LIN {X 0,Y 181.03,Z 246.971,A -85,B 0,C 180,E1 -24435.455,E2 -24435.455} C_VEL
LIN {X 0,Y 176.807,Z 236.449,A -85,B 0,C 180,E1 -24437.488,E2 -24437.488} C_VEL
LIN {X 0,Y 171.429,Z 226.879,A -85,B 0,C 180,E1 -24440.107,E2 -24440.107} C_VEL
LIN {X 0,Y 165.244,Z 217.098,A -85,B 0,C 180,E1 -24443.456,E2 -24443.456} C_VEL
LIN {X 0,Y 161.167,Z 211.387,A -85,B 0,C 180,E1 -24445.913,E2 -24445.913} C_VEL
LIN {X 0,Y 159.1,Z 208.478,A -85,B 0,C 180,E1 -24447.274,E2 -24447.274} C_VEL
LIN {X 0,Y 156.348,Z 204.614,A -85,B 0,C 180,E1 -24449.227,E2 -24449.227} C_VEL
LIN {X 0,Y 153.341,Z 201.146,A -85,B 0,C 180,E1 -24451.514,E2 -24451.514} C_VEL
LIN {X 0,Y 152.359,Z 199.454,A -85,B 0,C 180,E1 -24452.375,E2 -24452.375} C_VEL
LIN {X 0,Y 149.741,Z 197.177,A -85,B 0,C 180,E1 -24454.617,E2 -24454.617} C_VEL
LIN {X 0,Y 148.138,Z 194.255,A -85,B 0,C 180,E1 -24456.31,E2 -24456.31} C_VEL
LIN {X 0,Y 144.94,Z 191.854,A -85,B 0,C 180,E1 -24459.74,E2 -24459.74} C_VEL
LIN {X 0,Y 143.538,Z 189.332,A -85,B 0,C 180,E1 -24461.719,E2 -24461.719} C_VEL
LIN {X 0,Y 143.277,Z 188.126,A -85,B 0,C 180,E1 -24462.331,E2 -24462.331} C_VEL
LIN {X 0,Y 143.594,Z 188.094,A -85,B 0,C 180,E1 -24468.71,E2 -24468.71} C_VEL
LIN {X 0,Y 143.648,Z 188.066,A -85,B 0,C 180,E1 -24471.56,E2 -24471.56} C_VEL
LIN {X 0,Y 144.176,Z 188.004,A -85,B 0,C 180,E1 -24480,E2 -24480} C_VEL
LIN {X 0,Y 143.662,Z 188.078,A -85,B 0,C 180,E1 -24488.439,E2 -24488.439} C_VEL
LIN {X 0,Y 143.548,Z 188.085,A -85,B 0,C 180,E1 -24491.713,E2 -24491.713} C_VEL
LIN {X 0,Y 143.32,Z 188.307,A -85,B 0,C 180,E1 -24497.571,E2 -24497.571} C_VEL
LIN {X 0,Y 144.036,Z 190.441,A -85,B 0,C 180,E1 -24498.768,E2 -24498.768} C_VEL
LIN {X 0,Y 145.985,Z 192.88,A -85,B 0,C 180,E1 -24501.212,E2 -24501.212} C_VEL
LIN {X 0,Y 148.135,Z 194.263,A -85,B 0,C 180,E1 -24503.412,E2 -24503.412} C_VEL
LIN {X 0,Y 149.748,Z 197.216,A -85,B 0,C 180,E1 -24505.117,E2 -24505.117} C_VEL
LIN {X 0,Y 152.642,Z 199.935,A -85,B 0,C 180,E1 -24507.6,E2 -24507.6} C_VEL
LIN {X 0,Y 155.021,Z 203.316,A -85,B 0,C 180,E1 -24509.54,E2 -24509.54} C_VEL
LIN {X 0,Y 156.51,Z 204.938,A -85,B 0,C 180,E1 -24510.626,E2 -24510.626} C_VEL
LIN {X 0,Y 159.237,Z 208.646,A -85,B 0,C 180,E1 -24512.541,E2 -24512.541} C_VEL
LIN {X 0,Y 163.139,Z 214.191,A -85,B 0,C 180,E1 -24515.036,E2 -24515.036} C_VEL
LIN {X 0,Y 167.839,Z 222.521,A -85,B 0,C 180,E1 -24517.824,E2 -24517.824} C_VEL
LIN {X 0,Y 173.152,Z 233.173,A -85,B 0,C 180,E1 -24520.69,E2 -24520.69} C_VEL
LIN {X 0,Y 177.841,Z 244.163,A -85,B 0,C 180,E1 -24523.048,E2 -24523.048} C_VEL
LIN {X 0,Y 180.687,Z 252.004,A -85,B 0,C 180,E1 -24524.437,E2 -24524.437} C_VEL
LIN {X 0,Y 177.831,Z 293.742,A -85,B 0,C 180,E1 -24525.922,E2 -24525.922} C_VEL
LIN {X 0,Y 175.936,Z 307.466,A -85,B 0,C 180,E1 -24526.785,E2 -24526.785} C_VEL
LIN {X 0,Y 173.137,Z 320.253,A -85,B 0,C 180,E1 -24527.951,E2 -24527.951} C_VEL
LIN {X 0,Y 170.092,Z 331.321,A -85,B 0,C 180,E1 -24529.401,E2 -24529.401} C_VEL
LIN {X 0,Y 166.225,Z 342.868,A -85,B 0,C 180,E1 -24531.419,E2 -24531.419} C_VEL
LIN {X 0,Y 162.061,Z 353.267,A -85,B 0,C 180,E1 -24533.782,E2 -24533.782} C_VEL
LIN {X 0,Y 158.257,Z 361.771,A -85,B 0,C 180,E1 -24536.282,E2 -24536.282} C_VEL
LIN {X 0,Y 154.431,Z 369.618,A -85,B 0,C 180,E1 -24539.205,E2 -24539.205} C_VEL
LIN {X 0,Y 150.632,Z 377.289,A -85,B 0,C 180,E1 -24542.942,E2 -24542.942} C_VEL
LIN {X 0,Y 147.705,Z 382.545,A -85,B 0,C 180,E1 -24546.144,E2 -24546.144} C_VEL
LIN {X 0,Y 144.889,Z 387.639,A -85,B 0,C 180,E1 -24550.151,E2 -24550.151} C_VEL
LIN {X 0,Y 142.783,Z 391.597,A -85,B 0,C 180,E1 -24554.293,E2 -24554.293} C_VEL
LIN {X 0,Y 141.413,Z 394.526,A -85,B 0,C 180,E1 -24558.534,E2 -24558.534} C_VEL
LIN {X 0,Y 140.977,Z 395.483,A -85,B 0,C 180,E1 -24560.494,E2 -24560.494} C_VEL
LIN {X 0,Y 139.998,Z 396.49,A -85,B 0,C 180,E1 -24562.836,E2 -24562.836} C_VEL
LIN {X 0,Y 138.274,Z 397.195,A -85,B 0,C 180,E1 -24565.163,E2 -24565.163} C_VEL
LIN {X 0,Y 134.529,Z 397.679,A -85,B 0,C 180,E1 -24569.953,E2 -24569.953} C_VEL
LIN {X 0,Y 133.387,Z 397.283,A -85,B 0,C 180,E1 -24573.332,E2 -24573.332} C_VEL
LIN {X 0,Y 133.825,Z 395.721,A -85,B 0,C 180,E1 -24579.065,E2 -24579.065} C_VEL
LIN {X 0,Y 134.448,Z 394.311,A -85,B 0,C 180,E1 -24582.069,E2 -24582.069} C_VEL
LIN {X 0,Y 135.916,Z 391.36,A -85,B 0,C 180,E1 -24586.523,E2 -24586.523} C_VEL
LIN {X 0,Y 138.197,Z 387.373,A -85,B 0,C 180,E1 -24590.854,E2 -24590.854} C_VEL
LIN {X 0,Y 141.775,Z 381.247,A -85,B 0,C 180,E1 -24595.706,E2 -24595.706} C_VEL
LIN {X 0,Y 145.188,Z 375.115,A -85,B 0,C 180,E1 -24599.389,E2 -24599.389} C_VEL
LIN {X 0,Y 149.884,Z 366.268,A -85,B 0,C 180,E1 -24603.432,E2 -24603.432} C_VEL
LIN {X 0,Y 154.105,Z 357.763,A -85,B 0,C 180,E1 -24606.361,E2 -24606.361} C_VEL
LIN {X 0,Y 158.747,Z 347.258,A -85,B 0,C 180,E1 -24609.114,E2 -24609.114} C_VEL
LIN {X 0,Y 162.671,Z 336.859,A -85,B 0,C 180,E1 -24611.213,E2 -24611.213} C_VEL
LIN {X 0,Y 166.329,Z 325.448,A -85,B 0,C 180,E1 -24612.948,E2 -24612.948} C_VEL
LIN {X 0,Y 169.314,Z 313.676,A -85,B 0,C 180,E1 -24614.256,E2 -24614.256} C_VEL
LIN {X 0,Y 171.836,Z 300.262,A -85,B 0,C 180,E1 -24615.267,E2 -24615.267} C_VEL
LIN {X 0,Y 173.244,Z 287.392,A -85,B 0,C 180,E1 -24615.892,E2 -24615.892} C_VEL
LIN {X 0,Y 175.458,Z 253.977,A -85,B 0,C 180,E1 -24617.083,E2 -24617.083} C_VEL
LIN {X 0,Y 171.919,Z 244.299,A -85,B 0,C 180,E1 -24618.956,E2 -24618.956} C_VEL
LIN {X 0,Y 167.154,Z 233.408,A -85,B 0,C 180,E1 -24621.586,E2 -24621.586} C_VEL
LIN {X 0,Y 161.636,Z 222.544,A -85,B 0,C 180,E1 -24624.917,E2 -24624.917} C_VEL
LIN {X 0,Y 158.79,Z 217.886,A -85,B 0,C 180,E1 -24626.77,E2 -24626.77} C_VEL
LIN {X 0,Y 156.09,Z 214.087,A -85,B 0,C 180,E1 -24628.629,E2 -24628.629} C_VEL
LIN {X 0,Y 153.177,Z 210.078,A -85,B 0,C 180,E1 -24630.824,E2 -24630.824} C_VEL
LIN {X 0,Y 150.453,Z 206.422,A -85,B 0,C 180,E1 -24633.097,E2 -24633.097} C_VEL
LIN {X 0,Y 146.976,Z 202.464,A -85,B 0,C 180,E1 -24636.346,E2 -24636.346} C_VEL
LIN {X 0,Y 146.09,Z 200.68,A -85,B 0,C 180,E1 -24637.365,E2 -24637.365} C_VEL
LIN {X 0,Y 143.581,Z 198.76,A -85,B 0,C 180,E1 -24640.149,E2 -24640.149} C_VEL
LIN {X 0,Y 141.921,Z 195.955,A -85,B 0,C 180,E1 -24642.529,E2 -24642.529} C_VEL
LIN {X 0,Y 141.624,Z 195.129,A -85,B 0,C 180,E1 -24643.05,E2 -24643.05} C_VEL
LIN {X 0,Y 138.553,Z 193.165,A -85,B 0,C 180,E1 -24648.294,E2 -24648.294} C_VEL
LIN {X 0,Y 136.676,Z 189.596,A -85,B 0,C 180,E1 -24654.56,E2 -24654.56} C_VEL
LIN {X 0,Y 136.615,Z 188.962,A -85,B 0,C 180,E1 -24655.574,E2 -24655.574} C_VEL
LIN {X 0,Y 137.133,Z 188.886,A -85,B 0,C 180,E1 -24660,E2 -24660} C_VEL
LIN {X 0,Y 136.607,Z 189.164,A -85,B 0,C 180,E1 -24665.258,E2 -24665.258} C_VEL
LIN {X 0,Y 137.905,Z 192.426,A -85,B 0,C 180,E1 -24670.511,E2 -24670.511} C_VEL
LIN {X 0,Y 140.236,Z 194.528,A -85,B 0,C 180,E1 -24675.255,E2 -24675.255} C_VEL
LIN {X 0,Y 141.682,Z 195.221,A -85,B 0,C 180,E1 -24677.408,E2 -24677.408} C_VEL
LIN {X 0,Y 142.943,Z 197.948,A -85,B 0,C 180,E1 -24679.383,E2 -24679.383} C_VEL
LIN {X 0,Y 145.47,Z 200.379,A -85,B 0,C 180,E1 -24682.375,E2 -24682.375} C_VEL
LIN {X 0,Y 146.306,Z 201.102,A -85,B 0,C 180,E1 -24683.254,E2 -24683.254} C_VEL
LIN {X 0,Y 148.442,Z 204.412,A -85,B 0,C 180,E1 -24685.488,E2 -24685.488} C_VEL
LIN {X 0,Y 150.462,Z 206.34,A -85,B 0,C 180,E1 -24687.267,E2 -24687.267} C_VEL
LIN {X 0,Y 153.113,Z 210.035,A -85,B 0,C 180,E1 -24689.496,E2 -24689.496} C_VEL
LIN {X 0,Y 154.457,Z 211.806,A -85,B 0,C 180,E1 -24690.532,E2 -24690.532} C_VEL
LIN {X 0,Y 157.768,Z 216.391,A -85,B 0,C 180,E1 -24692.907,E2 -24692.907} C_VEL
LIN {X 0,Y 162.507,Z 223.419,A -85,B 0,C 180,E1 -24695.946,E2 -24695.946} C_VEL
LIN {X 0,Y 168.46,Z 233.167,A -85,B 0,C 180,E1 -24699.318,E2 -24699.318} C_VEL
LIN {X 0,Y 172.955,Z 241.65,A -85,B 0,C 180,E1 -24701.638,E2 -24701.638} C_VEL
LIN {X 0,Y 175.777,Z 248.785,A -85,B 0,C 180,E1 -24703.09,E2 -24703.09} C_VEL
LIN {X 0,Y 173.198,Z 286.39,A -85,B 0,C 180,E1 -24704.45,E2 -24704.45} C_VEL
LIN {X 0,Y 171.57,Z 298.932,A -85,B 0,C 180,E1 -24705.182,E2 -24705.182} C_VEL
LIN {X 0,Y 169.598,Z 309.113,A -85,B 0,C 180,E1 -24706.044,E2 -24706.044} C_VEL
LIN {X 0,Y 166.538,Z 321.437,A -85,B 0,C 180,E1 -24707.53,E2 -24707.53} C_VEL
LIN {X 0,Y 162.551,Z 333.931,A -85,B 0,C 180,E1 -24709.569,E2 -24709.569} C_VEL
LIN {X 0,Y 158.275,Z 344.869,A -85,B 0,C 180,E1 -24711.968,E2 -24711.968} C_VEL
LIN {X 0,Y 154.323,Z 353.759,A -85,B 0,C 180,E1 -24714.504,E2 -24714.504} C_VEL
LIN {X 0,Y 149.744,Z 363.2,A -85,B 0,C 180,E1 -24718.025,E2 -24718.025} C_VEL
LIN {X 0,Y 145.433,Z 371.074,A -85,B 0,C 180,E1 -24721.89,E2 -24721.89} C_VEL
LIN {X 0,Y 141.15,Z 378.13,A -85,B 0,C 180,E1 -24726.526,E2 -24726.526} C_VEL
LIN {X 0,Y 138.333,Z 382.823,A -85,B 0,C 180,E1 -24730.717,E2 -24730.717} C_VEL
LIN {X 0,Y 136.174,Z 386.413,A -85,B 0,C 180,E1 -24735.045,E2 -24735.045} C_VEL
LIN {X 0,Y 135.149,Z 388.264,A -85,B 0,C 180,E1 -24737.994,E2 -24737.994} C_VEL
LIN {X 0,Y 134.36,Z 389.654,A -85,B 0,C 180,E1 -24740.972,E2 -24740.972} C_VEL
LIN {X 0,Y 133.876,Z 390.643,A -85,B 0,C 180,E1 -24743.973,E2 -24743.973} C_VEL
LIN {X 0,Y 133.603,Z 391.249,A -85,B 0,C 180,E1 -24746.985,E2 -24746.985} C_VEL
LIN {X 0,Y 133.533,Z 391.476,A -85,B 0,C 180,E1 -24750,E2 -24750} C_VEL
LIN {X 0,Y 133.603,Z 391.28,A -85,B 0,C 180,E1 -24753.015,E2 -24753.015} C_VEL
LIN {X 0,Y 133.875,Z 390.693,A -85,B 0,C 180,E1 -24756.027,E2 -24756.027} C_VEL
LIN {X 0,Y 135.1,Z 388.365,A -85,B 0,C 180,E1 -24762.01,E2 -24762.01} C_VEL
LIN {X 0,Y 136.776,Z 385.492,A -85,B 0,C 180,E1 -24766.416,E2 -24766.416} C_VEL
LIN {X 0,Y 139.189,Z 381.594,A -85,B 0,C 180,E1 -24770.698,E2 -24770.698} C_VEL
LIN {X 0,Y 142.246,Z 376.564,A -85,B 0,C 180,E1 -24774.832,E2 -24774.832} C_VEL
LIN {X 0,Y 146.063,Z 370.224,A -85,B 0,C 180,E1 -24778.761,E2 -24778.761} C_VEL
LIN {X 0,Y 150.013,Z 362.842,A -85,B 0,C 180,E1 -24782.307,E2 -24782.307} C_VEL
LIN {X 0,Y 154.251,Z 354.218,A -85,B 0,C 180,E1 -24785.515,E2 -24785.515} C_VEL
LIN {X 0,Y 158.648,Z 344.353,A -85,B 0,C 180,E1 -24788.33,E2 -24788.33} C_VEL
LIN {X 0,Y 162.954,Z 333.238,A -85,B 0,C 180,E1 -24790.716,E2 -24790.716} C_VEL
LIN {X 0,Y 166.502,Z 322.34,A -85,B 0,C 180,E1 -24792.482,E2 -24792.482} C_VEL
LIN {X 0,Y 169.525,Z 310.294,A -85,B 0,C 180,E1 -24793.979,E2 -24793.979} C_VEL
LIN {X 0,Y 171.801,Z 298.279,A -85,B 0,C 180,E1 -24795.04,E2 -24795.04} C_VEL
LIN {X 0,Y 173.505,Z 284.761,A -85,B 0,C 180,E1 -24795.771,E2 -24795.771} C_VEL
LIN {X 0,Y 175.905,Z 248.819,A -85,B 0,C 180,E1 -24797.077,E2 -24797.077} C_VEL
LIN {X 0,Y 172.155,Z 239.744,A -85,B 0,C 180,E1 -24799.007,E2 -24799.007} C_VEL
LIN {X 0,Y 166.416,Z 229.505,A -85,B 0,C 180,E1 -24802.048,E2 -24802.048} C_VEL
LIN {X 0,Y 159.757,Z 219.039,A -85,B 0,C 180,E1 -24806.062,E2 -24806.062} C_VEL
LIN {X 0,Y 156.199,Z 214.146,A -85,B 0,C 180,E1 -24808.485,E2 -24808.485} C_VEL
LIN {X 0,Y 153.246,Z 210.087,A -85,B 0,C 180,E1 -24810.725,E2 -24810.725} C_VEL
LIN {X 0,Y 150.599,Z 206.524,A -85,B 0,C 180,E1 -24812.952,E2 -24812.952} C_VEL
LIN {X 0,Y 149.506,Z 205.392,A -85,B 0,C 180,E1 -24813.91,E2 -24813.91} C_VEL
LIN {X 0,Y 146.889,Z 202.243,A -85,B 0,C 180,E1 -24816.471,E2 -24816.471} C_VEL
LIN {X 0,Y 146.124,Z 200.675,A -85,B 0,C 180,E1 -24817.37,E2 -24817.37} C_VEL
LIN {X 0,Y 143.389,Z 198.517,A -85,B 0,C 180,E1 -24820.494,E2 -24820.494} C_VEL
LIN {X 0,Y 141.761,Z 195.483,A -85,B 0,C 180,E1 -24822.973,E2 -24822.973} C_VEL
LIN {X 0,Y 141.504,Z 194.987,A -85,B 0,C 180,E1 -24823.406,E2 -24823.406} C_VEL
LIN {X 0,Y 138.724,Z 193.315,A -85,B 0,C 180,E1 -24828.308,E2 -24828.308} C_VEL
LIN {X 0,Y 136.766,Z 189.75,A -85,B 0,C 180,E1 -24835.394,E2 -24835.394} C_VEL
LIN {X 0,Y 136.726,Z 188.939,A -85,B 0,C 180,E1 -24836.685,E2 -24836.685} C_VEL
LIN {X 0,Y 137.133,Z 188.88,A -85,B 0,C 180,E1 -24840,E2 -24840} C_VEL
LIN {X 0,Y 136.724,Z 189.067,A -85,B 0,C 180,E1 -24843.592,E2 -24843.592} C_VEL
LIN {X 0,Y 137.15,Z 191.005,A -85,B 0,C 180,E1 -24846.621,E2 -24846.621} C_VEL
LIN {X 0,Y 140.321,Z 194.528,A -85,B 0,C 180,E1 -24854.503,E2 -24854.503} C_VEL
LIN {X 0,Y 141.671,Z 195.155,A -85,B 0,C 180,E1 -24856.573,E2 -24856.573} C_VEL
LIN {X 0,Y 143.199,Z 198.264,A -85,B 0,C 180,E1 -24858.974,E2 -24858.974} C_VEL
LIN {X 0,Y 145.842,Z 200.558,A -85,B 0,C 180,E1 -24862.069,E2 -24862.069} C_VEL
LIN {X 0,Y 146.46,Z 201.426,A -85,B 0,C 180,E1 -24862.761,E2 -24862.761} C_VEL
LIN {X 0,Y 148.612,Z 204.553,A -85,B 0,C 180,E1 -24865.003,E2 -24865.003} C_VEL
LIN {X 0,Y 150.452,Z 206.304,A -85,B 0,C 180,E1 -24866.639,E2 -24866.639} C_VEL
LIN {X 0,Y 153.217,Z 210.087,A -85,B 0,C 180,E1 -24868.979,E2 -24868.979} C_VEL
LIN {X 0,Y 154.542,Z 211.92,A -85,B 0,C 180,E1 -24870.016,E2 -24870.016} C_VEL
LIN {X 0,Y 157.736,Z 216.284,A -85,B 0,C 180,E1 -24872.321,E2 -24872.321} C_VEL
LIN {X 0,Y 160.242,Z 220.06,A -85,B 0,C 180,E1 -24874,E2 -24874} C_VEL
LIN {X 0,Y 164.999,Z 228.872,A -85,B 0,C 180,E1 -24876.992,E2 -24876.992} C_VEL
LIN {X 0,Y 169.996,Z 239.495,A -85,B 0,C 180,E1 -24879.852,E2 -24879.852} C_VEL
LIN {X 0,Y 173.985,Z 249.452,A -85,B 0,C 180,E1 -24881.997,E2 -24881.997} C_VEL
LIN {X 0,Y 175.638,Z 254.083,A -85,B 0,C 180,E1 -24882.862,E2 -24882.862} C_VEL
LIN {X 0,Y 172.796,Z 293.594,A -85,B 0,C 180,E1 -24884.282,E2 -24884.282} C_VEL
LIN {X 0,Y 170.935,Z 306.77,A -85,B 0,C 180,E1 -24885.115,E2 -24885.115} C_VEL
LIN {X 0,Y 168.193,Z 318.996,A -85,B 0,C 180,E1 -24886.206,E2 -24886.206} C_VEL
LIN {X 0,Y 164.771,Z 331.164,A -85,B 0,C 180,E1 -24887.795,E2 -24887.795} C_VEL
LIN {X 0,Y 160.714,Z 342.71,A -85,B 0,C 180,E1 -24889.834,E2 -24889.834} C_VEL
LIN {X 0,Y 156.37,Z 353.108,A -85,B 0,C 180,E1 -24892.239,E2 -24892.239} C_VEL
LIN {X 0,Y 152.381,Z 361.611,A -85,B 0,C 180,E1 -24894.795,E2 -24894.795} C_VEL
LIN {X 0,Y 148.366,Z 369.458,A -85,B 0,C 180,E1 -24897.798,E2 -24897.798} C_VEL
LIN {X 0,Y 144.316,Z 377.128,A -85,B 0,C 180,E1 -24901.653,E2 -24901.653} C_VEL
LIN {X 0,Y 141.199,Z 382.383,A -85,B 0,C 180,E1 -24904.971,E2 -24904.971} C_VEL
LIN {X 0,Y 138.197,Z 387.477,A -85,B 0,C 180,E1 -24909.146,E2 -24909.146} C_VEL
LIN {X 0,Y 135.916,Z 391.435,A -85,B 0,C 180,E1 -24913.477,E2 -24913.477} C_VEL
LIN {X 0,Y 134.448,Z 394.364,A -85,B 0,C 180,E1 -24917.931,E2 -24917.931} C_VEL
LIN {X 0,Y 133.461,Z 396.754,A -85,B 0,C 180,E1 -24923.955,E2 -24923.955} C_VEL
LIN {X 0,Y 133.397,Z 397.363,A -85,B 0,C 180,E1 -24926.98,E2 -24926.98} C_VEL
LIN {X 0,Y 133.474,Z 397.575,A -85,B 0,C 180,E1 -24930,E2 -24930} C_VEL
LIN {X 0,Y 133.387,Z 397.283,A -85,B 0,C 180,E1 -24933.332,E2 -24933.332} C_VEL
LIN {X 0,Y 132.767,Z 396.787,A -85,B 0,C 180,E1 -24935.846,E2 -24935.846} C_VEL
LIN {X 0,Y 130.425,Z 395.377,A -85,B 0,C 180,E1 -24939.996,E2 -24939.996} C_VEL
LIN {X 0,Y 128.809,Z 393.752,A -85,B 0,C 180,E1 -24943.377,E2 -24943.377} C_VEL
LIN {X 0,Y 128.598,Z 392.23,A -85,B 0,C 180,E1 -24945.933,E2 -24945.933} C_VEL
LIN {X 0,Y 128.83,Z 391.648,A -85,B 0,C 180,E1 -24946.773,E2 -24946.773} C_VEL
LIN {X 0,Y 131.56,Z 387.209,A -85,B 0,C 180,E1 -24951.959,E2 -24951.959} C_VEL
LIN {X 0,Y 135.406,Z 381.083,A -85,B 0,C 180,E1 -24957.01,E2 -24957.01} C_VEL
LIN {X 0,Y 139.259,Z 374.519,A -85,B 0,C 180,E1 -24961.065,E2 -24961.065} C_VEL
LIN {X 0,Y 143.99,Z 366.103,A -85,B 0,C 180,E1 -24964.995,E2 -24964.995} C_VEL
LIN {X 0,Y 148.441,Z 357.598,A -85,B 0,C 180,E1 -24967.988,E2 -24967.988} C_VEL
LIN {X 0,Y 153.303,Z 347.092,A -85,B 0,C 180,E1 -24970.789,E2 -24970.789} C_VEL
LIN {X 0,Y 157.4,Z 336.693,A -85,B 0,C 180,E1 -24972.916,E2 -24972.916} C_VEL
LIN {X 0,Y 161.208,Z 325.28,A -85,B 0,C 180,E1 -24974.667,E2 -24974.667} C_VEL
LIN {X 0,Y 164.304,Z 313.506,A -85,B 0,C 180,E1 -24975.984,E2 -24975.984} C_VEL
LIN {X 0,Y 166.923,Z 300.053,A -85,B 0,C 180,E1 -24977,E2 -24977} C_VEL
LIN {X 0,Y 168.362,Z 287.367,A -85,B 0,C 180,E1 -24977.622,E2 -24977.622} C_VEL
LIN {X 0,Y 170.445,Z 255.864,A -85,B 0,C 180,E1 -24978.798,E2 -24978.798} C_VEL
LIN {X 0,Y 166.912,Z 246.185,A -85,B 0,C 180,E1 -24980.832,E2 -24980.832} C_VEL
LIN {X 0,Y 161.948,Z 234.865,A -85,B 0,C 180,E1 -24983.848,E2 -24983.848} C_VEL
LIN {X 0,Y 157.233,Z 225.737,A -85,B 0,C 180,E1 -24986.992,E2 -24986.992} C_VEL
LIN {X 0,Y 153.715,Z 220.288,A -85,B 0,C 180,E1 -24989.54,E2 -24989.54} C_VEL
LIN {X 0,Y 150.71,Z 216.148,A -85,B 0,C 180,E1 -24991.932,E2 -24991.932} C_VEL
LIN {X 0,Y 147.698,Z 212.016,A -85,B 0,C 180,E1 -24994.643,E2 -24994.643} C_VEL
LIN {X 0,Y 144.972,Z 208.712,A -85,B 0,C 180,E1 -24997.41,E2 -24997.41} C_VEL
LIN {X 0,Y 144.058,Z 207.206,A -85,B 0,C 180,E1 -24998.491,E2 -24998.491} C_VEL
LIN {X 0,Y 141.419,Z 204.613,A -85,B 0,C 180,E1 -25001.764,E2 -25001.764} C_VEL
LIN {X 0,Y 140.073,Z 201.884,A -85,B 0,C 180,E1 -25003.981,E2 -25003.981} C_VEL
LIN {X 0,Y 137.459,Z 200.096,A -85,B 0,C 180,E1 -25008.745,E2 -25008.745} C_VEL
LIN {X 0,Y 135.689,Z 196.502,A -85,B 0,C 180,E1 -25015.172,E2 -25015.172} C_VEL
LIN {X 0,Y 135.553,Z 195.943,A -85,B 0,C 180,E1 -25016.284,E2 -25016.284} C_VEL
LIN {X 0,Y 135.266,Z 195.729,A -85,B 0,C 180,E1 -25020,E2 -25020} C_VEL
LIN {X 0,Y 135.631,Z 196.097,A -85,B 0,C 180,E1 -25024.644,E2 -25024.644} C_VEL
LIN {X 0,Y 137.076,Z 199.648,A -85,B 0,C 180,E1 -25030.676,E2 -25030.676} C_VEL
LIN {X 0,Y 139.398,Z 201.612,A -85,B 0,C 180,E1 -25035.349,E2 -25035.349} C_VEL
LIN {X 0,Y 140.228,Z 202.188,A -85,B 0,C 180,E1 -25036.656,E2 -25036.656} C_VEL
LIN {X 0,Y 141.882,Z 205.241,A -85,B 0,C 180,E1 -25039.251,E2 -25039.251} C_VEL
LIN {X 0,Y 144.449,Z 207.667,A -85,B 0,C 180,E1 -25042.322,E2 -25042.322} C_VEL
LIN {X 0,Y 147.027,Z 211.417,A -85,B 0,C 180,E1 -25045.102,E2 -25045.102} C_VEL
LIN {X 0,Y 148.452,Z 212.923,A -85,B 0,C 180,E1 -25046.423,E2 -25046.423} C_VEL
LIN {X 0,Y 151.204,Z 216.674,A -85,B 0,C 180,E1 -25048.832,E2 -25048.832} C_VEL
LIN {X 0,Y 155.241,Z 222.527,A -85,B 0,C 180,E1 -25051.957,E2 -25051.957} C_VEL
LIN {X 0,Y 159.738,Z 229.506,A -85,B 0,C 180,E1 -25055.015,E2 -25055.015} C_VEL
LIN {X 0,Y 165.065,Z 238.564,A -85,B 0,C 180,E1 -25058.221,E2 -25058.221} C_VEL
LIN {X 0,Y 169.016,Z 246.239,A -85,B 0,C 180,E1 -25060.399,E2 -25060.399} C_VEL
LIN {X 0,Y 170.895,Z 251.125,A -85,B 0,C 180,E1 -25061.445,E2 -25061.445} C_VEL
LIN {X 0,Y 168.18,Z 287.683,A -85,B 0,C 180,E1 -25062.769,E2 -25062.769} C_VEL
LIN {X 0,Y 166.248,Z 300.852,A -85,B 0,C 180,E1 -25063.582,E2 -25063.582} C_VEL
LIN {X 0,Y 163.533,Z 313.81,A -85,B 0,C 180,E1 -25064.838,E2 -25064.838} C_VEL
LIN {X 0,Y 160.348,Z 325.096,A -85,B 0,C 180,E1 -25066.345,E2 -25066.345} C_VEL
LIN {X 0,Y 156.222,Z 336.722,A -85,B 0,C 180,E1 -25068.428,E2 -25068.428} C_VEL
LIN {X 0,Y 151.784,Z 347.168,A -85,B 0,C 180,E1 -25070.885,E2 -25070.885} C_VEL
LIN {X 0,Y 147.722,Z 355.7,A -85,B 0,C 180,E1 -25073.509,E2 -25073.509} C_VEL
LIN {X 0,Y 143.643,Z 363.602,A -85,B 0,C 180,E1 -25076.628,E2 -25076.628} C_VEL
LIN {X 0,Y 139.21,Z 371.238,A -85,B 0,C 180,E1 -25080.513,E2 -25080.513} C_VEL
LIN {X 0,Y 134.661,Z 378.294,A -85,B 0,C 180,E1 -25085.322,E2 -25085.322} C_VEL
LIN {X 0,Y 131.646,Z 382.987,A -85,B 0,C 180,E1 -25089.696,E2 -25089.696} C_VEL
LIN {X 0,Y 129.324,Z 386.576,A -85,B 0,C 180,E1 -25094.233,E2 -25094.233} C_VEL
LIN {X 0,Y 128.213,Z 388.427,A -85,B 0,C 180,E1 -25097.334,E2 -25097.334} C_VEL
LIN {X 0,Y 127.364,Z 389.817,A -85,B 0,C 180,E1 -25100.471,E2 -25100.471} C_VEL
LIN {X 0,Y 126.824,Z 390.805,A -85,B 0,C 180,E1 -25103.637,E2 -25103.637} C_VEL
LIN {X 0,Y 126.515,Z 391.411,A -85,B 0,C 180,E1 -25106.815,E2 -25106.815} C_VEL
LIN {X 0,Y 126.447,Z 391.637,A -85,B 0,C 180,E1 -25110,E2 -25110} C_VEL
LIN {X 0,Y 126.515,Z 391.442,A -85,B 0,C 180,E1 -25113.184,E2 -25113.184} C_VEL
LIN {X 0,Y 126.823,Z 390.854,A -85,B 0,C 180,E1 -25116.363,E2 -25116.363} C_VEL
LIN {X 0,Y 127.354,Z 389.886,A -85,B 0,C 180,E1 -25119.529,E2 -25119.529} C_VEL
LIN {X 0,Y 128.147,Z 388.527,A -85,B 0,C 180,E1 -25122.672,E2 -25122.672} C_VEL
LIN {X 0,Y 129.968,Z 385.654,A -85,B 0,C 180,E1 -25127.302,E2 -25127.302} C_VEL
LIN {X 0,Y 132.545,Z 381.755,A -85,B 0,C 180,E1 -25131.787,E2 -25131.787} C_VEL
LIN {X 0,Y 135.837,Z 376.725,A -85,B 0,C 180,E1 -25136.089,E2 -25136.089} C_VEL
LIN {X 0,Y 139.872,Z 370.385,A -85,B 0,C 180,E1 -25140.163,E2 -25140.163} C_VEL
LIN {X 0,Y 144.568,Z 361.976,A -85,B 0,C 180,E1 -25144.265,E2 -25144.265} C_VEL
LIN {X 0,Y 149.425,Z 352.598,A -85,B 0,C 180,E1 -25147.693,E2 -25147.693} C_VEL
LIN {X 0,Y 154.131,Z 342.235,A -85,B 0,C 180,E1 -25150.524,E2 -25150.524} C_VEL
LIN {X 0,Y 158.697,Z 330.548,A -85,B 0,C 180,E1 -25152.913,E2 -25152.913} C_VEL
LIN {X 0,Y 162.403,Z 318.876,A -85,B 0,C 180,E1 -25154.686,E2 -25154.686} C_VEL
LIN {X 0,Y 165.267,Z 306.733,A -85,B 0,C 180,E1 -25156.076,E2 -25156.076} C_VEL
LIN {X 0,Y 167.643,Z 293.48,A -85,B 0,C 180,E1 -25157.077,E2 -25157.077} C_VEL
LIN {X 0,Y 169.009,Z 280.763,A -85,B 0,C 180,E1 -25157.649,E2 -25157.649} C_VEL
LIN {X 0,Y 171.083,Z 251.356,A -85,B 0,C 180,E1 -25158.693,E2 -25158.693} C_VEL
LIN {X 0,Y 167.902,Z 243.673,A -85,B 0,C 180,E1 -25160.455,E2 -25160.455} C_VEL
LIN {X 0,Y 162.371,Z 233.72,A -85,B 0,C 180,E1 -25163.617,E2 -25163.617} C_VEL
LIN {X 0,Y 156.754,Z 224.61,A -85,B 0,C 180,E1 -25167.27,E2 -25167.27} C_VEL
LIN {X 0,Y 153.383,Z 219.801,A -85,B 0,C 180,E1 -25169.733,E2 -25169.733} C_VEL
LIN {X 0,Y 150.898,Z 216.252,A -85,B 0,C 180,E1 -25171.75,E2 -25171.75} C_VEL
LIN {X 0,Y 147.819,Z 212.101,A -85,B 0,C 180,E1 -25174.531,E2 -25174.531} C_VEL
LIN {X 0,Y 145.049,Z 208.729,A -85,B 0,C 180,E1 -25177.375,E2 -25177.375} C_VEL
LIN {X 0,Y 144.113,Z 207.191,A -85,B 0,C 180,E1 -25178.497,E2 -25178.497} C_VEL
LIN {X 0,Y 141.42,Z 204.571,A -85,B 0,C 180,E1 -25181.904,E2 -25181.904} C_VEL
LIN {X 0,Y 140.193,Z 201.964,A -85,B 0,C 180,E1 -25183.995,E2 -25183.995} C_VEL
LIN {X 0,Y 137.432,Z 199.976,A -85,B 0,C 180,E1 -25189.282,E2 -25189.282} C_VEL
LIN {X 0,Y 135.775,Z 196.369,A -85,B 0,C 180,E1 -25196.476,E2 -25196.476} C_VEL
LIN {X 0,Y 135.755,Z 195.954,A -85,B 0,C 180,E1 -25197.032,E2 -25197.032} C_VEL
LIN {X 0,Y 135.65,Z 195.904,A -85,B 0,C 180,E1 -25201.484,E2 -25201.484} C_VEL
LIN {X 0,Y 135.788,Z 196.37,A -85,B 0,C 180,E1 -25203.338,E2 -25203.338} C_VEL
LIN {X 0,Y 137.416,Z 199.96,A -85,B 0,C 180,E1 -25210.403,E2 -25210.403} C_VEL
LIN {X 0,Y 140.232,Z 202.125,A -85,B 0,C 180,E1 -25215.814,E2 -25215.814} C_VEL
LIN {X 0,Y 142.08,Z 205.432,A -85,B 0,C 180,E1 -25218.755,E2 -25218.755} C_VEL
LIN {X 0,Y 144.492,Z 207.705,A -85,B 0,C 180,E1 -25221.675,E2 -25221.675} C_VEL
LIN {X 0,Y 146.779,Z 211.095,A -85,B 0,C 180,E1 -25224.204,E2 -25224.204} C_VEL
LIN {X 0,Y 148.493,Z 212.967,A -85,B 0,C 180,E1 -25225.83,E2 -25225.83} C_VEL
LIN {X 0,Y 151.964,Z 217.777,A -85,B 0,C 180,E1 -25228.863,E2 -25228.863} C_VEL
LIN {X 0,Y 155.153,Z 222.337,A -85,B 0,C 180,E1 -25231.319,E2 -25231.319} C_VEL
LIN {X 0,Y 157.449,Z 226.01,A -85,B 0,C 180,E1 -25232.961,E2 -25232.961} C_VEL
LIN {X 0,Y 161.72,Z 234.27,A -85,B 0,C 180,E1 -25235.831,E2 -25235.831} C_VEL
LIN {X 0,Y 166.453,Z 244.787,A -85,B 0,C 180,E1 -25238.733,E2 -25238.733} C_VEL
LIN {X 0,Y 170.609,Z 255.899,A -85,B 0,C 180,E1 -25241.133,E2 -25241.133} C_VEL
LIN {X 0,Y 170.274,Z 262.497,A -85,B 0,C 180,E1 -25241.417,E2 -25241.417} C_VEL
LIN {X 0,Y 167.85,Z 293.997,A -85,B 0,C 180,E1 -25242.577,E2 -25242.577} C_VEL
LIN {X 0,Y 165.784,Z 307.675,A -85,B 0,C 180,E1 -25243.467,E2 -25243.467} C_VEL
LIN {X 0,Y 162.873,Z 319.941,A -85,B 0,C 180,E1 -25244.604,E2 -25244.604} C_VEL
LIN {X 0,Y 159.04,Z 332.59,A -85,B 0,C 180,E1 -25246.333,E2 -25246.333} C_VEL
LIN {X 0,Y 154.867,Z 343.846,A -85,B 0,C 180,E1 -25248.418,E2 -25248.418} C_VEL
LIN {X 0,Y 150.33,Z 353.98,A -85,B 0,C 180,E1 -25250.867,E2 -25250.867} C_VEL
LIN {X 0,Y 145.747,Z 363.117,A -85,B 0,C 180,E1 -25253.794,E2 -25253.794} C_VEL
LIN {X 0,Y 140.776,Z 372.164,A -85,B 0,C 180,E1 -25257.627,E2 -25257.627} C_VEL
LIN {X 0,Y 136.768,Z 379.207,A -85,B 0,C 180,E1 -25261.624,E2 -25261.624} C_VEL
LIN {X 0,Y 133.642,Z 384.041,A -85,B 0,C 180,E1 -25265.121,E2 -25265.121} C_VEL
LIN {X 0,Y 130.626,Z 388.746,A -85,B 0,C 180,E1 -25269.53,E2 -25269.53} C_VEL
LIN {X 0,Y 128.499,Z 392.346,A -85,B 0,C 180,E1 -25274.13,E2 -25274.13} C_VEL
LIN {X 0,Y 127.478,Z 394.202,A -85,B 0,C 180,E1 -25277.26,E2 -25277.26} C_VEL
LIN {X 0,Y 126.404,Z 396.592,A -85,B 0,C 180,E1 -25283.616,E2 -25283.616} C_VEL
LIN {X 0,Y 126.302,Z 397.201,A -85,B 0,C 180,E1 -25286.81,E2 -25286.81} C_VEL
LIN {X 0,Y 126.389,Z 397.414,A -85,B 0,C 180,E1 -25290,E2 -25290} C_VEL
LIN {X 0,Y 126.3,Z 397.164,A -85,B 0,C 180,E1 -25293.294,E2 -25293.294} C_VEL
LIN {X 0,Y 126.795,Z 395.558,A -85,B 0,C 180,E1 -25299.572,E2 -25299.572} C_VEL
LIN {X 0,Y 127.478,Z 394.148,A -85,B 0,C 180,E1 -25302.74,E2 -25302.74} C_VEL
LIN {X 0,Y 128.83,Z 391.648,A -85,B 0,C 180,E1 -25306.773,E2 -25306.773} C_VEL
LIN {X 0,Y 129.278,Z 389.82,A -85,B 0,C 180,E1 -25309.26,E2 -25309.26} C_VEL
LIN {X 0,Y 128.833,Z 386.331,A -85,B 0,C 180,E1 -25313.376,E2 -25313.376} C_VEL
LIN {X 0,Y 128.948,Z 382.174,A -85,B 0,C 180,E1 -25317.375,E2 -25317.375} C_VEL
LIN {X 0,Y 130.23,Z 379.284,A -85,B 0,C 180,E1 -25319.585,E2 -25319.585} C_VEL
LIN {X 0,Y 134.051,Z 372.994,A -85,B 0,C 180,E1 -25323.401,E2 -25323.401} C_VEL
LIN {X 0,Y 139.124,Z 364.343,A -85,B 0,C 180,E1 -25327.315,E2 -25327.315} C_VEL
LIN {X 0,Y 143.88,Z 355.48,A -85,B 0,C 180,E1 -25330.332,E2 -25330.332} C_VEL
LIN {X 0,Y 149.004,Z 344.568,A -85,B 0,C 180,E1 -25333.15,E2 -25333.15} C_VEL
LIN {X 0,Y 153.35,Z 333.535,A -85,B 0,C 180,E1 -25335.264,E2 -25335.264} C_VEL
LIN {X 0,Y 157.389,Z 321.17,A -85,B 0,C 180,E1 -25336.987,E2 -25336.987} C_VEL
LIN {X 0,Y 160.39,Z 309.434,A -85,B 0,C 180,E1 -25338.151,E2 -25338.151} C_VEL
LIN {X 0,Y 162.667,Z 296.575,A -85,B 0,C 180,E1 -25339.021,E2 -25339.021} C_VEL
LIN {X 0,Y 164.282,Z 278.871,A -85,B 0,C 180,E1 -25339.756,E2 -25339.756} C_VEL
LIN {X 0,Y 165.691,Z 257.995,A -85,B 0,C 180,E1 -25340.557,E2 -25340.557} C_VEL
LIN {X 0,Y 162.083,Z 248.197,A -85,B 0,C 180,E1 -25342.819,E2 -25342.819} C_VEL
LIN {X 0,Y 157.784,Z 238.319,A -85,B 0,C 180,E1 -25345.685,E2 -25345.685} C_VEL
LIN {X 0,Y 153.622,Z 229.978,A -85,B 0,C 180,E1 -25348.737,E2 -25348.737} C_VEL
LIN {X 0,Y 148.777,Z 222.714,A -85,B 0,C 180,E1 -25352.671,E2 -25352.671} C_VEL
LIN {X 0,Y 145.518,Z 218.257,A -85,B 0,C 180,E1 -25355.763,E2 -25355.763} C_VEL
LIN {X 0,Y 142.886,Z 214.684,A -85,B 0,C 180,E1 -25358.677,E2 -25358.677} C_VEL
LIN {X 0,Y 142.021,Z 213.606,A -85,B 0,C 180,E1 -25359.733,E2 -25359.733} C_VEL
LIN {X 0,Y 139.501,Z 210.567,A -85,B 0,C 180,E1 -25363.237,E2 -25363.237} C_VEL
LIN {X 0,Y 138.555,Z 208.679,A -85,B 0,C 180,E1 -25364.932,E2 -25364.932} C_VEL
LIN {X 0,Y 136.035,Z 206.618,A -85,B 0,C 180,E1 -25370.087,E2 -25370.087} C_VEL
LIN {X 0,Y 134.68,Z 203.063,A -85,B 0,C 180,E1 -25376.26,E2 -25376.26} C_VEL
LIN {X 0,Y 134.423,Z 202.875,A -85,B 0,C 180,E1 -25381.498,E2 -25381.498} C_VEL
LIN {X 0,Y 134.689,Z 203.255,A -85,B 0,C 180,E1 -25384.302,E2 -25384.302} C_VEL
LIN {X 0,Y 136.665,Z 207.41,A -85,B 0,C 180,E1 -25391.871,E2 -25391.871} C_VEL
LIN {X 0,Y 138.779,Z 209.009,A -85,B 0,C 180,E1 -25395.832,E2 -25395.832} C_VEL
LIN {X 0,Y 140.703,Z 212.335,A -85,B 0,C 180,E1 -25398.946,E2 -25398.946} C_VEL
LIN {X 0,Y 142.748,Z 214.412,A -85,B 0,C 180,E1 -25401.512,E2 -25401.512} C_VEL
LIN {X 0,Y 145.367,Z 218.107,A -85,B 0,C 180,E1 -25404.455,E2 -25404.455} C_VEL
LIN {X 0,Y 146.591,Z 219.677,A -85,B 0,C 180,E1 -25405.67,E2 -25405.67} C_VEL
LIN {X 0,Y 149.819,Z 224.322,A -85,B 0,C 180,E1 -25408.61,E2 -25408.61} C_VEL
LIN {X 0,Y 153.244,Z 229.448,A -85,B 0,C 180,E1 -25411.351,E2 -25411.351} C_VEL
LIN {X 0,Y 158.36,Z 237.812,A -85,B 0,C 180,E1 -25414.945,E2 -25414.945} C_VEL
LIN {X 0,Y 163.764,Z 247.851,A -85,B 0,C 180,E1 -25418.287,E2 -25418.287} C_VEL
LIN {X 0,Y 166.028,Z 253.23,A -85,B 0,C 180,E1 -25419.632,E2 -25419.632} C_VEL
LIN {X 0,Y 164.336,Z 278.285,A -85,B 0,C 180,E1 -25420.594,E2 -25420.594} C_VEL
LIN {X 0,Y 162.832,Z 292.836,A -85,B 0,C 180,E1 -25421.21,E2 -25421.21} C_VEL
LIN {X 0,Y 160.523,Z 305.58,A -85,B 0,C 180,E1 -25422.136,E2 -25422.136} C_VEL
LIN {X 0,Y 157.475,Z 318.037,A -85,B 0,C 180,E1 -25423.512,E2 -25423.512} C_VEL
LIN {X 0,Y 153.674,Z 329.986,A -85,B 0,C 180,E1 -25425.32,E2 -25425.32} C_VEL
LIN {X 0,Y 149.417,Z 340.634,A -85,B 0,C 180,E1 -25427.457,E2 -25427.457} C_VEL
LIN {X 0,Y 144.877,Z 350.343,A -85,B 0,C 180,E1 -25430.002,E2 -25430.002} C_VEL
LIN {X 0,Y 140.324,Z 359.172,A -85,B 0,C 180,E1 -25433.058,E2 -25433.058} C_VEL
LIN {X 0,Y 135.391,Z 367.782,A -85,B 0,C 180,E1 -25436.972,E2 -25436.972} C_VEL
LIN {X 0,Y 130.903,Z 374.65,A -85,B 0,C 180,E1 -25441.106,E2 -25441.106} C_VEL
LIN {X 0,Y 127.087,Z 380.148,A -85,B 0,C 180,E1 -25445.496,E2 -25445.496} C_VEL
LIN {X 0,Y 124.065,Z 384.459,A -85,B 0,C 180,E1 -25450.13,E2 -25450.13} C_VEL
LIN {X 0,Y 122.508,Z 386.739,A -85,B 0,C 180,E1 -25453.331,E2 -25453.331} C_VEL
LIN {X 0,Y 121.28,Z 388.59,A -85,B 0,C 180,E1 -25456.597,E2 -25456.597} C_VEL
LIN {X 0,Y 120.355,Z 389.98,A -85,B 0,C 180,E1 -25459.911,E2 -25459.911} C_VEL
LIN {X 0,Y 119.768,Z 390.967,A -85,B 0,C 180,E1 -25463.26,E2 -25463.26} C_VEL
LIN {X 0,Y 119.44,Z 391.574,A -85,B 0,C 180,E1 -25466.627,E2 -25466.627} C_VEL
LIN {X 0,Y 119.363,Z 391.799,A -85,B 0,C 180,E1 -25470,E2 -25470} C_VEL
LIN {X 0,Y 119.439,Z 391.603,A -85,B 0,C 180,E1 -25473.373,E2 -25473.373} C_VEL
LIN {X 0,Y 119.766,Z 391.016,A -85,B 0,C 180,E1 -25476.74,E2 -25476.74} C_VEL
LIN {X 0,Y 121.227,Z 388.689,A -85,B 0,C 180,E1 -25483.409,E2 -25483.409} C_VEL
LIN {X 0,Y 123.201,Z 385.816,A -85,B 0,C 180,E1 -25488.285,E2 -25488.285} C_VEL
LIN {X 0,Y 125.955,Z 381.917,A -85,B 0,C 180,E1 -25492.991,E2 -25492.991} C_VEL
LIN {X 0,Y 129.502,Z 376.885,A -85,B 0,C 180,E1 -25497.47,E2 -25497.47} C_VEL
LIN {X 0,Y 133.773,Z 370.545,A -85,B 0,C 180,E1 -25501.693,E2 -25501.693} C_VEL
LIN {X 0,Y 138.871,Z 361.95,A -85,B 0,C 180,E1 -25505.995,E2 -25505.995} C_VEL
LIN {X 0,Y 143.875,Z 352.757,A -85,B 0,C 180,E1 -25509.421,E2 -25509.421} C_VEL
LIN {X 0,Y 148.82,Z 342.393,A -85,B 0,C 180,E1 -25512.295,E2 -25512.295} C_VEL
LIN {X 0,Y 153.583,Z 330.705,A -85,B 0,C 180,E1 -25514.713,E2 -25514.713} C_VEL
LIN {X 0,Y 157.431,Z 319.032,A -85,B 0,C 180,E1 -25516.504,E2 -25516.504} C_VEL
LIN {X 0,Y 160.422,Z 306.887,A -85,B 0,C 180,E1 -25517.904,E2 -25517.904} C_VEL
LIN {X 0,Y 162.884,Z 293.736,A -85,B 0,C 180,E1 -25518.896,E2 -25518.896} C_VEL
LIN {X 0,Y 164.339,Z 280.563,A -85,B 0,C 180,E1 -25519.489,E2 -25519.489} C_VEL
LIN {X 0,Y 166.308,Z 253.624,A -85,B 0,C 180,E1 -25520.46,E2 -25520.46} C_VEL
LIN {X 0,Y 163.842,Z 247.753,A -85,B 0,C 180,E1 -25521.93,E2 -25521.93} C_VEL
LIN {X 0,Y 158.018,Z 237.044,A -85,B 0,C 180,E1 -25525.565,E2 -25525.565} C_VEL
LIN {X 0,Y 153.073,Z 229.053,A -85,B 0,C 180,E1 -25529.093,E2 -25529.093} C_VEL
LIN {X 0,Y 148.853,Z 222.685,A -85,B 0,C 180,E1 -25532.591,E2 -25532.591} C_VEL
LIN {X 0,Y 145.731,Z 218.409,A -85,B 0,C 180,E1 -25535.574,E2 -25535.574} C_VEL
LIN {X 0,Y 142.958,Z 214.698,A -85,B 0,C 180,E1 -25538.667,E2 -25538.667} C_VEL
LIN {X 0,Y 142.253,Z 213.701,A -85,B 0,C 180,E1 -25539.553,E2 -25539.553} C_VEL
LIN {X 0,Y 139.651,Z 210.742,A -85,B 0,C 180,E1 -25543.18,E2 -25543.18} C_VEL
LIN {X 0,Y 138.692,Z 208.739,A -85,B 0,C 180,E1 -25544.947,E2 -25544.947} C_VEL
LIN {X 0,Y 135.91,Z 206.331,A -85,B 0,C 180,E1 -25551.075,E2 -25551.075} C_VEL
LIN {X 0,Y 134.819,Z 202.967,A -85,B 0,C 180,E1 -25557.759,E2 -25557.759} C_VEL
LIN {X 0,Y 134.834,Z 203.05,A -85,B 0,C 180,E1 -25562.24,E2 -25562.24} C_VEL
LIN {X 0,Y 137.024,Z 207.652,A -85,B 0,C 180,E1 -25571.612,E2 -25571.612} C_VEL
LIN {X 0,Y 138.881,Z 209.043,A -85,B 0,C 180,E1 -25575.125,E2 -25575.125} C_VEL
LIN {X 0,Y 140.602,Z 212.132,A -85,B 0,C 180,E1 -25578.016,E2 -25578.016} C_VEL
LIN {X 0,Y 142.718,Z 214.263,A -85,B 0,C 180,E1 -25580.746,E2 -25580.746} C_VEL
LIN {X 0,Y 145.134,Z 217.786,A -85,B 0,C 180,E1 -25583.547,E2 -25583.547} C_VEL
LIN {X 0,Y 146.494,Z 219.396,A -85,B 0,C 180,E1 -25584.915,E2 -25584.915} C_VEL
LIN {X 0,Y 149.801,Z 224.193,A -85,B 0,C 180,E1 -25587.979,E2 -25587.979} C_VEL
LIN {X 0,Y 153.828,Z 230.201,A -85,B 0,C 180,E1 -25591.201,E2 -25591.201} C_VEL
LIN {X 0,Y 157.953,Z 238.477,A -85,B 0,C 180,E1 -25594.237,E2 -25594.237} C_VEL
LIN {X 0,Y 162.498,Z 248.919,A -85,B 0,C 180,E1 -25597.265,E2 -25597.265} C_VEL
